   LaserEnd_Ext()
   LIN {X 9.720, Y 7.023, Z 94.350}
   LaserStart_Ext()
   LIN {X 9.720, Y -22.180, Z 94.350}
   LaserEnd_Ext()
   LIN {X 10.720, Y -19.592, Z 94.350}
   LaserStart_Ext()
   LIN {X 10.720, Y 0.002, Z 94.350}
   LaserEnd_Ext()
   LIN {X 5.886, Y -14.219, Z 95.200}
   LaserStart_Ext()
   LIN {X 6.069, Y -14.305, Z 95.200} C_DIS
   LIN {X 6.222, Y -14.503, Z 95.200} C_DIS
   LIN {X 7.618, Y -16.321, Z 95.200} C_DIS
   LIN {X 7.985, Y -18.449, Z 95.200} C_DIS
   LIN {X 7.977, Y -18.559, Z 95.200} C_DIS
   LIN {X 7.385, Y -20.644, Z 95.200} C_DIS
   LIN {X 5.903, Y -22.320, Z 95.200} C_DIS
   LIN {X 5.822, Y -22.379, Z 95.200} C_DIS
   LIN {X 3.889, Y -23.196, Z 95.200} C_DIS
   LIN {X 2.561, Y -23.174, Z 95.200} C_DIS
   LIN {X 1.827, Y -23.160, Z 95.200} C_DIS
   LIN {X 0.884, Y -22.715, Z 95.200} C_DIS
   LIN {X -0.043, Y -22.280, Z 95.200} C_DIS
   LIN {X -0.599, Y -21.642, Z 95.200} C_DIS
   LIN {X -1.407, Y -20.706, Z 95.200} C_DIS
   LIN {X -1.753, Y -19.527, Z 95.200} C_DIS
   LIN {X -1.997, Y -18.705, Z 95.200} C_DIS
   LIN {X -1.693, Y -17.374, Z 95.200} C_DIS
   LIN {X -1.338, Y -15.799, Z 95.200} C_DIS
   LIN {X -0.761, Y -15.153, Z 95.200} C_DIS
   LIN {X 0.076, Y -14.226, Z 95.200} C_DIS
   LIN {X 1.728, Y -13.494, Z 95.200} C_DIS
   LIN {X 1.983, Y -13.382, Z 95.200} C_DIS
   LIN {X 2.192, Y -13.383, Z 95.200} C_DIS
   LIN {X 4.149, Y -13.393, Z 95.200} C_DIS
   LIN {X 5.886, Y -14.219, Z 95.200}
   LaserEnd_Ext()
   LIN {X -5.498, Y -20.746, Z 95.200}
   LaserStart_Ext()
   LIN {X -6.019, Y -18.561, Z 95.200} C_DIS
   LIN {X -5.683, Y -16.347, Z 95.200} C_DIS
   LIN {X -5.539, Y -15.427, Z 95.200} C_DIS
   LIN {X -5.305, Y -14.701, Z 95.200} C_DIS
   LIN {X -4.631, Y -12.568, Z 95.200} C_DIS
   LIN {X -3.664, Y -8.937, Z 95.200} C_DIS
   LIN {X -3.638, Y -8.835, Z 95.200} C_DIS
   LIN {X -2.885, Y -5.203, Z 95.200} C_DIS
   LIN {X -2.566, Y -3.350, Z 95.200} C_DIS
   LIN {X -2.304, Y -1.628, Z 95.200} C_DIS
   LIN {X -2.221, Y -0.926, Z 95.200} C_DIS
   LIN {X -2.134, Y -0.229, Z 95.200} C_DIS
   LIN {X -1.879, Y 2.505, Z 95.200} C_DIS
   LIN {X -1.732, Y 6.473, Z 95.200} C_DIS
   LIN {X -1.751, Y 11.457, Z 95.200} C_DIS
   LIN {X -2.156, Y 15.764, Z 95.200} C_DIS
   LIN {X -3.665, Y 24.816, Z 95.200} C_DIS
   LIN {X -3.882, Y 25.807, Z 95.200} C_DIS
   LIN {X -4.262, Y 27.109, Z 95.200} C_DIS
   LIN {X -5.179, Y 30.344, Z 95.200} C_DIS
   LIN {X -6.003, Y 32.721, Z 95.200} C_DIS
   LIN {X -6.559, Y 34.208, Z 95.200} C_DIS
   LIN {X -7.213, Y 35.871, Z 95.200} C_DIS
   LIN {X -7.302, Y 36.098, Z 95.200} C_DIS
   LIN {X -7.368, Y 36.249, Z 95.200} C_DIS
   LIN {X -8.249, Y 38.271, Z 95.200} C_DIS
   LIN {X -8.844, Y 39.539, Z 95.200} C_DIS
   LIN {X -8.928, Y 39.719, Z 95.200} C_DIS
   LIN {X -9.034, Y 39.937, Z 95.200} C_DIS
   LIN {X -9.471, Y 40.846, Z 95.200} C_DIS
   LIN {X -9.752, Y 41.728, Z 95.200} C_DIS
   LIN {X -9.875, Y 42.116, Z 95.200} C_DIS
   LIN {X -9.856, Y 42.526, Z 95.200} C_DIS
   LIN {X -9.820, Y 43.494, Z 95.200} C_DIS
   LIN {X -9.382, Y 44.438, Z 95.200} C_DIS
   LIN {X -9.073, Y 45.084, Z 95.200} C_DIS
   LIN {X -8.537, Y 45.414, Z 95.200} C_DIS
   LIN {X -6.714, Y 46.543, Z 95.200} C_DIS
   LIN {X -6.039, Y 46.527, Z 95.200} C_DIS
   LIN {X -4.970, Y 46.499, Z 95.200} C_DIS
   LIN {X -3.550, Y 45.789, Z 95.200} C_DIS
   LIN {X -3.415, Y 45.721, Z 95.200} C_DIS
   LIN {X -2.455, Y 44.605, Z 95.200} C_DIS
   LIN {X -1.797, Y 43.427, Z 95.200} C_DIS
   LIN {X -1.731, Y 43.308, Z 95.200} C_DIS
   LIN {X -1.605, Y 43.078, Z 95.200} C_DIS
   LIN {X -0.809, Y 41.619, Z 95.200} C_DIS
   LIN {X -0.065, Y 40.182, Z 95.200} C_DIS
   LIN {X 0.629, Y 38.834, Z 95.200} C_DIS
   LIN {X 0.808, Y 38.450, Z 95.200} C_DIS
   LIN {X 3.585, Y 32.416, Z 95.200} C_DIS
   LIN {X 4.111, Y 31.131, Z 95.200} C_DIS
   LIN {X 5.388, Y 27.470, Z 95.200} C_DIS
   LIN {X 6.945, Y 23.293, Z 95.200} C_DIS
   LIN {X 7.649, Y 21.147, Z 95.200} C_DIS
   LIN {X 9.644, Y 13.265, Z 95.200} C_DIS
   LIN {X 9.975, Y 11.963, Z 95.200} C_DIS
   LIN {X 10.184, Y 10.632, Z 95.200} C_DIS
   LIN {X 11.571, Y 2.143, Z 95.200} C_DIS
   LIN {X 11.760, Y 0.223, Z 95.200} C_DIS
   LIN {X 12.012, Y -2.890, Z 95.200} C_DIS
   LIN {X 12.109, Y -4.088, Z 95.200} C_DIS
   LIN {X 12.241, Y -7.692, Z 95.200} C_DIS
   LIN {X 12.287, Y -8.871, Z 95.200} C_DIS
   LIN {X 12.289, Y -9.206, Z 95.200} C_DIS
   LIN {X 12.281, Y -12.675, Z 95.200} C_DIS
   LIN {X 12.228, Y -14.437, Z 95.200} C_DIS
   LIN {X 12.185, Y -15.633, Z 95.200} C_DIS
   LIN {X 12.037, Y -18.085, Z 95.200} C_DIS
   LIN {X 11.990, Y -18.889, Z 95.200} C_DIS
   LIN {X 11.897, Y -19.276, Z 95.200} C_DIS
   LIN {X 11.284, Y -21.766, Z 95.200} C_DIS
   LIN {X 9.658, Y -24.025, Z 95.200} C_DIS
   LIN {X 8.896, Y -25.053, Z 95.200} C_DIS
   LIN {X 5.588, Y -26.867, Z 95.200} C_DIS
   LIN {X 5.471, Y -26.932, Z 95.200} C_DIS
   LIN {X 5.278, Y -26.929, Z 95.200} C_DIS
   LIN {X -0.325, Y -26.687, Z 95.200} C_DIS
   LIN {X -1.234, Y -26.081, Z 95.200} C_DIS
   LIN {X -3.494, Y -24.588, Z 95.200} C_DIS
   LIN {X -4.454, Y -23.208, Z 95.200} C_DIS
   LIN {X -5.166, Y -22.172, Z 95.200} C_DIS
   LIN {X -5.498, Y -20.746, Z 95.200}
   LaserEnd_Ext()
   LIN {X -0.513, Y -25.360, Z 95.200}
   LaserStart_Ext()
   LIN {X 6.256, Y -25.360, Z 95.200}
   LaserEnd_Ext()
   LIN {X 8.080, Y -24.360, Z 95.200}
   LaserStart_Ext()
   LIN {X -2.025, Y -24.360, Z 95.200}
   LaserEnd_Ext()
   LIN {X -3.130, Y -23.360, Z 95.200}
   LaserStart_Ext()
   LIN {X -0.096, Y -23.360, Z 95.200}
   LaserEnd_Ext()
   LIN {X 6.069, Y -23.360, Z 95.200}
   LaserStart_Ext()
   LIN {X 8.904, Y -23.360, Z 95.200}
   LaserEnd_Ext()
   LIN {X 9.624, Y -22.360, Z 95.200}
   LaserStart_Ext()
   LIN {X 7.202, Y -22.360, Z 95.200}
   LaserEnd_Ext()
   LIN {X -1.299, Y -22.360, Z 95.200}
   LaserStart_Ext()
   LIN {X -3.823, Y -22.360, Z 95.200}
   LaserEnd_Ext()
   LIN {X -4.328, Y -21.360, Z 95.200}
   LaserStart_Ext()
   LIN {X -2.164, Y -21.360, Z 95.200}
   LaserEnd_Ext()
   LIN {X 8.087, Y -21.360, Z 95.200}
   LaserStart_Ext()
   LIN {X 10.344, Y -21.360, Z 95.200}
   LaserEnd_Ext()
   LIN {X 10.600, Y -20.360, Z 95.200}
   LaserStart_Ext()
   LIN {X 8.505, Y -20.360, Z 95.200}
   LaserEnd_Ext()
   LIN {X -2.551, Y -20.360, Z 95.200}
   LaserStart_Ext()
   LIN {X -4.562, Y -20.360, Z 95.200}
   LaserEnd_Ext()
   LIN {X -4.800, Y -19.360, Z 95.200}
   LaserStart_Ext()
   LIN {X -2.846, Y -19.360, Z 95.200}
   LaserEnd_Ext()
   LIN {X 8.789, Y -19.360, Z 95.200}
   LaserStart_Ext()
   LIN {X 10.847, Y -19.360, Z 95.200}
   LaserEnd_Ext()
   LIN {X 11.019, Y -18.360, Z 95.200}
   LaserStart_Ext()
   LIN {X 8.983, Y -18.360, Z 95.200}
   LaserEnd_Ext()
   LIN {X -2.944, Y -18.360, Z 95.200}
   LaserStart_Ext()
   LIN {X -4.977, Y -18.360, Z 95.200}
   LaserEnd_Ext()
   LIN {X -4.825, Y -17.360, Z 95.200}
   LaserStart_Ext()
   LIN {X -2.716, Y -17.360, Z 95.200}
   LaserEnd_Ext()
   LIN {X 8.812, Y -17.360, Z 95.200}
   LaserStart_Ext()
   LIN {X 11.079, Y -17.360, Z 95.200}
   LaserEnd_Ext()
   LIN {X 11.139, Y -16.360, Z 95.200}
   LaserStart_Ext()
   LIN {X 8.639, Y -16.360, Z 95.200}
   LaserEnd_Ext()
   LIN {X -2.489, Y -16.360, Z 95.200}
   LaserStart_Ext()
   LIN {X -4.673, Y -16.360, Z 95.200}
   LaserEnd_Ext()
   LIN {X -4.467, Y -15.360, Z 95.200}
   LaserStart_Ext()
   LIN {X -2.235, Y -15.360, Z 95.200}
   LaserEnd_Ext()
   LIN {X 8.140, Y -15.360, Z 95.200}
   LaserStart_Ext()
   LIN {X 11.194, Y -15.360, Z 95.200}
   LaserEnd_Ext()
   LIN {X 11.230, Y -14.360, Z 95.200}
   LaserStart_Ext()
   LIN {X 7.373, Y -14.360, Z 95.200}
   LaserEnd_Ext()
   LIN {X -1.392, Y -14.360, Z 95.200}
   LaserStart_Ext()
   LIN {X -4.149, Y -14.360, Z 95.200}
   LaserEnd_Ext()
   LIN {X -3.833, Y -13.360, Z 95.200}
   LaserStart_Ext()
   LIN {X -0.425, Y -13.360, Z 95.200}
   LaserEnd_Ext()
   LIN {X 6.409, Y -13.360, Z 95.200}
   LaserStart_Ext()
   LIN {X 11.260, Y -13.360, Z 95.200}
   LaserEnd_Ext()
   LIN {X 11.282, Y -12.360, Z 95.200}
   LaserStart_Ext()
   LIN {X -3.541, Y -12.360, Z 95.200}
   LaserEnd_Ext()
   LIN {X -3.274, Y -11.360, Z 95.200}
   LaserStart_Ext()
   LIN {X 11.284, Y -11.360, Z 95.200}
   LaserEnd_Ext()
   LIN {X 11.286, Y -10.360, Z 95.200}
   LaserStart_Ext()
   LIN {X -3.008, Y -10.360, Z 95.200}
   LaserEnd_Ext()
   LIN {X -2.742, Y -9.360, Z 95.200}
   LaserStart_Ext()
   LIN {X 11.289, Y -9.360, Z 95.200}
   LaserEnd_Ext()
   LIN {X 11.267, Y -8.360, Z 95.200}
   LaserStart_Ext()
   LIN {X -2.518, Y -8.360, Z 95.200}
   LaserEnd_Ext()
   LIN {X -2.311, Y -7.360, Z 95.200}
   LaserStart_Ext()
   LIN {X 11.228, Y -7.360, Z 95.200}
   LaserEnd_Ext()
   LIN {X 11.192, Y -6.360, Z 95.200}
   LaserStart_Ext()
   LIN {X -2.104, Y -6.360, Z 95.200}
   LaserEnd_Ext()
   LIN {X -1.897, Y -5.360, Z 95.200}
   LaserStart_Ext()
   LIN {X 11.155, Y -5.360, Z 95.200}
   LaserEnd_Ext()
   LIN {X 11.118, Y -4.360, Z 95.200}
   LaserStart_Ext()
   LIN {X -1.725, Y -4.360, Z 95.200}
   LaserEnd_Ext()
   LIN {X -1.556, Y -3.360, Z 95.200}
   LaserStart_Ext()
   LIN {X 11.047, Y -3.360, Z 95.200}
   LaserEnd_Ext()
   LIN {X 10.966, Y -2.360, Z 95.200}
   LaserStart_Ext()
   LIN {X -1.404, Y -2.360, Z 95.200}
   LaserEnd_Ext()
   LIN {X -1.265, Y -1.360, Z 95.200}
   LaserStart_Ext()
   LIN {X 10.885, Y -1.360, Z 95.200}
   LaserEnd_Ext()
   LIN {X 10.804, Y -0.360, Z 95.200}
   LaserStart_Ext()
   LIN {X -1.142, Y -0.360, Z 95.200}
   LaserEnd_Ext()
   LIN {X -1.048, Y 0.640, Z 95.200}
   LaserStart_Ext()
   LIN {X 10.714, Y 0.640, Z 95.200}
   LaserEnd_Ext()
   LIN {X 10.615, Y 1.640, Z 95.200}
   LaserStart_Ext()
   LIN {X -0.955, Y 1.640, Z 95.200}
   LaserEnd_Ext()
   LIN {X -0.873, Y 2.640, Z 95.200}
   LaserStart_Ext()
   LIN {X 10.476, Y 2.640, Z 95.200}
   LaserEnd_Ext()
   LIN {X 10.313, Y 3.640, Z 95.200}
   LaserStart_Ext()
   LIN {X -0.836, Y 3.640, Z 95.200}
   LaserEnd_Ext()
   LIN {X -0.799, Y 4.640, Z 95.200}
   LaserStart_Ext()
   LIN {X 10.150, Y 4.640, Z 95.200}
   LaserEnd_Ext()
   LIN {X 9.986, Y 5.640, Z 95.200}
   LaserStart_Ext()
   LIN {X -0.762, Y 5.640, Z 95.200}
   LaserEnd_Ext()
   LIN {X -0.733, Y 6.640, Z 95.200}
   LaserStart_Ext()
   LIN {X 9.823, Y 6.640, Z 95.200}
   LaserEnd_Ext()
   LIN {X 9.660, Y 7.640, Z 95.200}
   LaserStart_Ext()
   LIN {X -0.736, Y 7.640, Z 95.200}
   LaserEnd_Ext()
   LIN {X -0.740, Y 8.640, Z 95.200}
   LaserStart_Ext()
   LIN {X 9.496, Y 8.640, Z 95.200}
   LaserEnd_Ext()
   LIN {X 9.333, Y 9.640, Z 95.200}
   LaserStart_Ext()
   LIN {X -0.744, Y 9.640, Z 95.200}
   LaserEnd_Ext()
   LIN {X -0.748, Y 10.640, Z 95.200}
   LaserStart_Ext()
   LIN {X 9.171, Y 10.640, Z 95.200}
   LaserEnd_Ext()
   LIN {X 9.014, Y 11.640, Z 95.200}
   LaserStart_Ext()
   LIN {X -0.764, Y 11.640, Z 95.200}
   LaserEnd_Ext()
   LIN {X -0.858, Y 12.640, Z 95.200}
   LaserStart_Ext()
   LIN {X 8.771, Y 12.640, Z 95.200}
   LaserEnd_Ext()
   LIN {X 8.517, Y 13.640, Z 95.200}
   LaserStart_Ext()
   LIN {X -0.952, Y 13.640, Z 95.200}
   LaserEnd_Ext()
   LIN {X -1.046, Y 14.640, Z 95.200}
   LaserStart_Ext()
   LIN {X 8.264, Y 14.640, Z 95.200}
   LaserEnd_Ext()
   LIN {X 8.011, Y 15.640, Z 95.200}
   LaserStart_Ext()
   LIN {X -1.140, Y 15.640, Z 95.200}
   LaserEnd_Ext()
   LIN {X -1.288, Y 16.640, Z 95.200}
   LaserStart_Ext()
   LIN {X 7.758, Y 16.640, Z 95.200}
   LaserEnd_Ext()
   LIN {X 7.505, Y 17.640, Z 95.200}
   LaserStart_Ext()
   LIN {X -1.455, Y 17.640, Z 95.200}
   LaserEnd_Ext()
   LIN {X -1.622, Y 18.640, Z 95.200}
   LaserStart_Ext()
   LIN {X 7.252, Y 18.640, Z 95.200}
   LaserEnd_Ext()
   LIN {X 6.999, Y 19.640, Z 95.200}
   LaserStart_Ext()
   LIN {X -1.789, Y 19.640, Z 95.200}
   LaserEnd_Ext()
   LIN {X -1.955, Y 20.640, Z 95.200}
   LaserStart_Ext()
   LIN {X 6.746, Y 20.640, Z 95.200}
   LaserEnd_Ext()
   LIN {X 6.435, Y 21.640, Z 95.200}
   LaserStart_Ext()
   LIN {X -2.122, Y 21.640, Z 95.200}
   LaserEnd_Ext()
   LIN {X -2.289, Y 22.640, Z 95.200}
   LaserStart_Ext()
   LIN {X 6.106, Y 22.640, Z 95.200}
   LaserEnd_Ext()
   LIN {X 5.748, Y 23.640, Z 95.200}
   LaserStart_Ext()
   LIN {X -2.455, Y 23.640, Z 95.200}
   LaserEnd_Ext()
   LIN {X -2.622, Y 24.640, Z 95.200}
   LaserStart_Ext()
   LIN {X 5.375, Y 24.640, Z 95.200}
   LaserEnd_Ext()
   LIN {X 5.003, Y 25.640, Z 95.200}
   LaserStart_Ext()
   LIN {X -2.822, Y 25.640, Z 95.200}
   LaserEnd_Ext()
   LIN {X -3.083, Y 26.640, Z 95.200}
   LaserStart_Ext()
   LIN {X 4.630, Y 26.640, Z 95.200}
   LaserEnd_Ext()
   LIN {X 4.270, Y 27.640, Z 95.200}
   LaserStart_Ext()
   LIN {X -3.373, Y 27.640, Z 95.200}
   LaserEnd_Ext()
   LIN {X -3.657, Y 28.640, Z 95.200}
   LaserStart_Ext()
   LIN {X 3.921, Y 28.640, Z 95.200}
   LaserEnd_Ext()
   LIN {X 3.572, Y 29.640, Z 95.200}
   LaserStart_Ext()
   LIN {X -3.940, Y 29.640, Z 95.200}
   LaserEnd_Ext()
   LIN {X -4.225, Y 30.640, Z 95.200}
   LaserStart_Ext()
   LIN {X 3.224, Y 30.640, Z 95.200}
   LaserEnd_Ext()
   LIN {X 2.822, Y 31.640, Z 95.200}
   LaserStart_Ext()
   LIN {X -4.570, Y 31.640, Z 95.200}
   LaserEnd_Ext()
   LIN {X -4.917, Y 32.640, Z 95.200}
   LaserStart_Ext()
   LIN {X 2.381, Y 32.640, Z 95.200}
   LaserEnd_Ext()
   LIN {X 1.921, Y 33.640, Z 95.200}
   LaserStart_Ext()
   LIN {X -5.279, Y 33.640, Z 95.200}
   LaserEnd_Ext()
   LIN {X -5.654, Y 34.640, Z 95.200}
   LaserStart_Ext()
   LIN {X 1.461, Y 34.640, Z 95.200}
   LaserEnd_Ext()
   LIN {X 1.000, Y 35.640, Z 95.200}
   LaserStart_Ext()
   LIN {X -6.048, Y 35.640, Z 95.200}
   LaserEnd_Ext()
   LIN {X -6.447, Y 36.640, Z 95.200}
   LaserStart_Ext()
   LIN {X 0.540, Y 36.640, Z 95.200}
   LaserEnd_Ext()
   LIN {X 0.080, Y 37.640, Z 95.200}
   LaserStart_Ext()
   LIN {X -6.883, Y 37.640, Z 95.200}
   LaserEnd_Ext()
   LIN {X -7.319, Y 38.640, Z 95.200}
   LaserStart_Ext()
   LIN {X -0.396, Y 38.640, Z 95.200}
   LaserEnd_Ext()
   LIN {X -0.911, Y 39.640, Z 95.200}
   LaserStart_Ext()
   LIN {X -7.787, Y 39.640, Z 95.200}
   LaserEnd_Ext()
   LIN {X -8.262, Y 40.640, Z 95.200}
   LaserStart_Ext()
   LIN {X -1.428, Y 40.640, Z 95.200}
   LaserEnd_Ext()
   LIN {X -1.960, Y 41.640, Z 95.200}
   LaserStart_Ext()
   LIN {X -8.674, Y 41.640, Z 95.200}
   LaserEnd_Ext()
   LIN {X -8.851, Y 42.640, Z 95.200}
   LaserStart_Ext()
   LIN {X -2.506, Y 42.640, Z 95.200}
   LaserEnd_Ext()
   LIN {X -3.061, Y 43.640, Z 95.200}
   LaserStart_Ext()
   LIN {X -8.650, Y 43.640, Z 95.200}
   LaserEnd_Ext()
   LIN {X -7.888, Y 44.640, Z 95.200}
   LaserStart_Ext()
   LIN {X -3.803, Y 44.640, Z 95.200}
   LaserEnd_Ext()
   LIN {X 7.418, Y -20.676, Z 96.050}
   LaserStart_Ext()
   LIN {X 7.313, Y -20.795, Z 96.050} C_DIS
   LIN {X 5.955, Y -22.298, Z 96.050} C_DIS
   LIN {X 4.796, Y -22.790, Z 96.050} C_DIS
   LIN {X 3.975, Y -23.138, Z 96.050} C_DIS
   LIN {X 2.680, Y -23.116, Z 96.050} C_DIS
   LIN {X 1.920, Y -23.105, Z 96.050} C_DIS
   LIN {X 1.422, Y -22.874, Z 96.050} C_DIS
   LIN {X 0.048, Y -22.229, Z 96.050} C_DIS
   LIN {X -1.160, Y -20.841, Z 96.050} C_DIS
   LIN {X -1.320, Y -20.658, Z 96.050} C_DIS
   LIN {X -1.384, Y -20.446, Z 96.050} C_DIS
   LIN {X -1.914, Y -18.659, Z 96.050} C_DIS
   LIN {X -1.369, Y -16.270, Z 96.050} C_DIS
   LIN {X -1.243, Y -15.719, Z 96.050} C_DIS
   LIN {X -0.908, Y -15.348, Z 96.050} C_DIS
   LIN {X 0.156, Y -14.168, Z 96.050} C_DIS
   LIN {X 1.141, Y -13.732, Z 96.050} C_DIS
   LIN {X 2.053, Y -13.326, Z 96.050} C_DIS
   LIN {X 3.470, Y -13.328, Z 96.050} C_DIS
   LIN {X 4.219, Y -13.332, Z 96.050} C_DIS
   LIN {X 4.753, Y -13.586, Z 96.050} C_DIS
   LIN {X 6.141, Y -14.240, Z 96.050} C_DIS
   LIN {X 7.304, Y -15.743, Z 96.050} C_DIS
   LIN {X 7.695, Y -16.252, Z 96.050} C_DIS
   LIN {X 7.803, Y -16.879, Z 96.050} C_DIS
   LIN {X 8.076, Y -18.429, Z 96.050} C_DIS
   LIN {X 7.460, Y -20.527, Z 96.050} C_DIS
   LIN {X 7.418, Y -20.676, Z 96.050}
   LaserEnd_Ext()
   LIN {X -8.287, Y 38.272, Z 96.050}
   LaserStart_Ext()
   LIN {X -7.348, Y 36.132, Z 96.050} C_DIS
   LIN {X -6.974, Y 35.180, Z 96.050} C_DIS
   LIN {X -5.639, Y 31.611, Z 96.050} C_DIS
   LIN {X -5.201, Y 30.347, Z 96.050} C_DIS
   LIN {X -4.714, Y 28.628, Z 96.050} C_DIS
   LIN {X -3.924, Y 25.925, Z 96.050} C_DIS
   LIN {X -3.475, Y 23.867, Z 96.050} C_DIS
   LIN {X -2.206, Y 16.260, Z 96.050} C_DIS
   LIN {X -1.721, Y 11.097, Z 96.050} C_DIS
   LIN {X -1.704, Y 6.823, Z 96.050} C_DIS
   LIN {X -1.878, Y 2.146, Z 96.050} C_DIS
   LIN {X -2.093, Y -0.165, Z 96.050} C_DIS
   LIN {X -2.167, Y -0.755, Z 96.050} C_DIS
   LIN {X -2.285, Y -1.759, Z 96.050} C_DIS
   LIN {X -2.445, Y -2.806, Z 96.050} C_DIS
   LIN {X -2.997, Y -6.017, Z 96.050} C_DIS
   LIN {X -3.487, Y -8.375, Z 96.050} C_DIS
   LIN {X -3.992, Y -10.385, Z 96.050} C_DIS
   LIN {X -4.557, Y -12.506, Z 96.050} C_DIS
   LIN {X -5.255, Y -14.716, Z 96.050} C_DIS
   LIN {X -5.465, Y -15.389, Z 96.050} C_DIS
   LIN {X -5.553, Y -15.995, Z 96.050} C_DIS
   LIN {X -5.937, Y -18.524, Z 96.050} C_DIS
   LIN {X -5.120, Y -21.953, Z 96.050} C_DIS
   LIN {X -5.076, Y -22.134, Z 96.050} C_DIS
   LIN {X -4.986, Y -22.262, Z 96.050} C_DIS
   LIN {X -3.398, Y -24.545, Z 96.050} C_DIS
   LIN {X -0.974, Y -26.147, Z 96.050} C_DIS
   LIN {X -0.221, Y -26.638, Z 96.050} C_DIS
   LIN {X 0.213, Y -26.717, Z 96.050} C_DIS
   LIN {X 4.984, Y -26.957, Z 96.050} C_DIS
   LIN {X 5.688, Y -26.829, Z 96.050} C_DIS
   LIN {X 8.909, Y -25.025, Z 96.050} C_DIS
   LIN {X 9.026, Y -24.954, Z 96.050} C_DIS
   LIN {X 9.240, Y -24.652, Z 96.050} C_DIS
   LIN {X 11.374, Y -21.688, Z 96.050} C_DIS
   LIN {X 11.683, Y -20.434, Z 96.050} C_DIS
   LIN {X 12.072, Y -18.810, Z 96.050} C_DIS
   LIN {X 12.258, Y -15.609, Z 96.050} C_DIS
   LIN {X 12.263, Y -15.475, Z 96.050} C_DIS
   LIN {X 12.349, Y -12.595, Z 96.050} C_DIS
   LIN {X 12.354, Y -10.415, Z 96.050} C_DIS
   LIN {X 12.346, Y -8.791, Z 96.050} C_DIS
   LIN {X 12.172, Y -4.347, Z 96.050} C_DIS
   LIN {X 12.155, Y -3.988, Z 96.050} C_DIS
   LIN {X 11.862, Y -0.359, Z 96.050} C_DIS
   LIN {X 11.621, Y 2.083, Z 96.050} C_DIS
   LIN {X 10.107, Y 11.350, Z 96.050} C_DIS
   LIN {X 10.032, Y 11.811, Z 96.050} C_DIS
   LIN {X 9.888, Y 12.387, Z 96.050} C_DIS
   LIN {X 7.731, Y 20.909, Z 96.050} C_DIS
   LIN {X 6.836, Y 23.635, Z 96.050} C_DIS
   LIN {X 4.858, Y 28.942, Z 96.050} C_DIS
   LIN {X 4.054, Y 31.249, Z 96.050} C_DIS
   LIN {X 3.722, Y 32.059, Z 96.050} C_DIS
   LIN {X 1.159, Y 37.626, Z 96.050} C_DIS
   LIN {X 0.617, Y 38.806, Z 96.050} C_DIS
   LIN {X -0.122, Y 40.227, Z 96.050} C_DIS
   LIN {X -0.872, Y 41.675, Z 96.050} C_DIS
   LIN {X -1.122, Y 42.135, Z 96.050} C_DIS
   LIN {X -1.794, Y 43.357, Z 96.050} C_DIS
   LIN {X -2.507, Y 44.626, Z 96.050} C_DIS
   LIN {X -3.482, Y 45.765, Z 96.050} C_DIS
   LIN {X -4.742, Y 46.391, Z 96.050} C_DIS
   LIN {X -5.040, Y 46.539, Z 96.050} C_DIS
   LIN {X -5.608, Y 46.551, Z 96.050} C_DIS
   LIN {X -6.785, Y 46.578, Z 96.050} C_DIS
   LIN {X -7.367, Y 46.217, Z 96.050} C_DIS
   LIN {X -9.123, Y 45.135, Z 96.050} C_DIS
   LIN {X -9.539, Y 44.263, Z 96.050} C_DIS
   LIN {X -9.867, Y 43.593, Z 96.050} C_DIS
   LIN {X -9.904, Y 42.944, Z 96.050} C_DIS
   LIN {X -9.940, Y 42.181, Z 96.050} C_DIS
   LIN {X -9.722, Y 41.496, Z 96.050} C_DIS
   LIN {X -9.527, Y 40.875, Z 96.050} C_DIS
   LIN {X -9.344, Y 40.499, Z 96.050} C_DIS
   LIN {X -8.982, Y 39.749, Z 96.050} C_DIS
   LIN {X -8.308, Y 38.319, Z 96.050}
   LaserEnd_Ext()
   LIN {X 10.602, Y 2.117, Z 96.050}
   LaserStart_Ext()
   LIN {X 10.602, Y -20.641, Z 96.050}
   LaserEnd_Ext()
   LIN {X 9.602, Y -22.438, Z 96.050}
   LaserStart_Ext()
   LIN {X 9.602, Y 8.241, Z 96.050}
   LaserEnd_Ext()
   LIN {X 8.602, Y 13.391, Z 96.050}
   LaserStart_Ext()
   LIN {X 8.602, Y -15.834, Z 96.050}
   LaserEnd_Ext()
   LIN {X 8.602, Y -20.187, Z 96.050}
   LaserStart_Ext()
   LIN {X 8.602, Y -23.827, Z 96.050}
   LaserEnd_Ext()
   LIN {X 7.602, Y -24.611, Z 96.050}
   LaserStart_Ext()
   LIN {X 7.602, Y -21.966, Z 96.050}
   LaserEnd_Ext()
   LIN {X 7.602, Y -14.494, Z 96.050}
   LaserStart_Ext()
   LIN {X 7.602, Y 17.343, Z 96.050}
   LaserEnd_Ext()
   LIN {X 6.602, Y 21.142, Z 96.050}
   LaserStart_Ext()
   LIN {X 6.602, Y -13.353, Z 96.050}
   LaserEnd_Ext()
   LIN {X 6.602, Y -23.059, Z 96.050}
   LaserStart_Ext()
   LIN {X 6.602, Y -25.171, Z 96.050}
   LaserEnd_Ext()
   LIN {X 5.602, Y -25.732, Z 96.050}
   LaserStart_Ext()
   LIN {X 5.602, Y -23.534, Z 96.050}
   LaserEnd_Ext()
   LIN {X 5.602, Y -12.880, Z 96.050}
   LaserStart_Ext()
   LIN {X 5.602, Y 24.083, Z 96.050}
   LaserEnd_Ext()
   LIN {X 4.602, Y 26.766, Z 96.050}
   LaserStart_Ext()
   LIN {X 4.602, Y -12.410, Z 96.050}
   LaserEnd_Ext()
   LIN {X 4.602, Y -23.958, Z 96.050}
   LaserStart_Ext()
   LIN {X 4.602, Y -25.937, Z 96.050}
   LaserEnd_Ext()
   LIN {X 3.602, Y -25.887, Z 96.050}
   LaserStart_Ext()
   LIN {X 3.602, Y -24.132, Z 96.050}
   LaserEnd_Ext()
   LIN {X 3.602, Y -12.329, Z 96.050}
   LaserStart_Ext()
   LIN {X 3.602, Y 29.508, Z 96.050}
   LaserEnd_Ext()
   LIN {X 2.602, Y 32.101, Z 96.050}
   LaserStart_Ext()
   LIN {X 2.602, Y -12.327, Z 96.050}
   LaserEnd_Ext()
   LIN {X 2.602, Y -24.115, Z 96.050}
   LaserStart_Ext()
   LIN {X 2.602, Y -25.836, Z 96.050}
   LaserEnd_Ext()
   LIN {X 1.602, Y -25.786, Z 96.050}
   LaserStart_Ext()
   LIN {X 1.602, Y -24.053, Z 96.050}
   LaserEnd_Ext()
   LIN {X 1.602, Y -12.432, Z 96.050}
   LaserStart_Ext()
   LIN {X 1.602, Y 34.274, Z 96.050}
   LaserEnd_Ext()
   LIN {X 0.602, Y 36.446, Z 96.050}
   LaserStart_Ext()
   LIN {X 0.602, Y -12.877, Z 96.050}
   LaserEnd_Ext()
   LIN {X 0.602, Y -23.594, Z 96.050}
   LaserStart_Ext()
   LIN {X 0.602, Y -25.736, Z 96.050}
   LaserEnd_Ext()
   LIN {X -0.398, Y -25.329, Z 96.050}
   LaserStart_Ext()
   LIN {X -0.398, Y -23.123, Z 96.050}
   LaserEnd_Ext()
   LIN {X -0.398, Y -13.338, Z 96.050}
   LaserStart_Ext()
   LIN {X -0.398, Y 38.591, Z 96.050}
   LaserEnd_Ext()
   LIN {X -1.398, Y 40.517, Z 96.050}
   LaserStart_Ext()
   LIN {X -1.398, Y 17.492, Z 96.050}
   LaserEnd_Ext()
   LIN {X -1.398, Y -2.576, Z 96.050}
   LaserStart_Ext()
   LIN {X -1.398, Y -14.398, Z 96.050}
   LaserEnd_Ext()
   LIN {X -1.398, Y -22.091, Z 96.050}
   LaserStart_Ext()
   LIN {X -1.398, Y -24.668, Z 96.050}
   LaserEnd_Ext()
   LIN {X -2.398, Y -24.007, Z 96.050}
   LaserStart_Ext()
   LIN {X -2.398, Y -20.543, Z 96.050}
   LaserEnd_Ext()
   LIN {X -2.398, Y -16.286, Z 96.050}
   LaserStart_Ext()
   LIN {X -2.398, Y -8.051, Z 96.050}
   LaserEnd_Ext()
   LIN {X -2.398, Y 23.490, Z 96.050}
   LaserStart_Ext()
   LIN {X -2.398, Y 42.380, Z 96.050}
   LaserEnd_Ext()
   LIN {X -3.398, Y 44.137, Z 96.050}
   LaserStart_Ext()
   LIN {X -3.398, Y 27.691, Z 96.050}
   LaserEnd_Ext()
   LIN {X -3.398, Y -12.041, Z 96.050}
   LaserStart_Ext()
   LIN {X -3.398, Y -22.793, Z 96.050}
   LaserEnd_Ext()
   LIN {X -4.398, Y -20.667, Z 96.050}
   LaserStart_Ext()
   LIN {X -4.398, Y -15.327, Z 96.050}
   LaserEnd_Ext()
   LIN {X -4.398, Y 31.084, Z 96.050}
   LaserStart_Ext()
   LIN {X -4.398, Y 45.103, Z 96.050}
   LaserEnd_Ext()
   LIN {X -5.398, Y 45.546, Z 96.050}
   LaserStart_Ext()
   LIN {X -5.398, Y 33.822, Z 96.050}
   LaserEnd_Ext()
   LIN {X -6.398, Y 36.449, Z 96.050}
   LaserStart_Ext()
   LIN {X -6.398, Y 45.569, Z 96.050}
   LaserEnd_Ext()
   LIN {X -7.398, Y 45.023, Z 96.050}
   LaserStart_Ext()
   LIN {X -7.398, Y 38.733, Z 96.050}
   LaserEnd_Ext()
   LIN {X -8.398, Y 40.839, Z 96.050}
   LaserStart_Ext()
   LIN {X -8.398, Y 44.332, Z 96.050}
   LaserEnd_Ext()
   LIN {X 3.573, Y -13.273, Z 96.900}
   LaserStart_Ext()
   LIN {X 4.290, Y -13.271, Z 96.900} C_DIS
   LIN {X 5.074, Y -13.637, Z 96.900} C_DIS
   LIN {X 6.213, Y -14.174, Z 96.900} C_DIS
   LIN {X 7.100, Y -15.321, Z 96.900} C_DIS
   LIN {X 7.772, Y -16.183, Z 96.900} C_DIS
   LIN {X 7.933, Y -17.082, Z 96.900} C_DIS
   LIN {X 8.158, Y -18.359, Z 96.900} C_DIS
   LIN {X 7.838, Y -19.449, Z 96.900} C_DIS
   LIN {X 7.497, Y -20.622, Z 96.900} C_DIS
   LIN {X 6.714, Y -21.492, Z 96.900} C_DIS
   LIN {X 6.039, Y -22.238, Z 96.900} C_DIS
   LIN {X 4.614, Y -22.843, Z 96.900} C_DIS
   LIN {X 4.072, Y -23.077, Z 96.900} C_DIS
   LIN {X 3.668, Y -23.074, Z 96.900} C_DIS
   LIN {X 2.014, Y -23.049, Z 96.900} C_DIS
   LIN {X 0.291, Y -22.250, Z 96.900} C_DIS
   LIN {X 0.139, Y -22.178, Z 96.900} C_DIS
   LIN {X 0.006, Y -22.025, Z 96.900} C_DIS
   LIN {X -1.232, Y -20.610, Z 96.900} C_DIS
   LIN {X -1.728, Y -18.962, Z 96.900} C_DIS
   LIN {X -1.832, Y -18.612, Z 96.900} C_DIS
   LIN {X -1.725, Y -18.145, Z 96.900} C_DIS
   LIN {X -1.158, Y -15.655, Z 96.900} C_DIS
   LIN {X 0.155, Y -14.202, Z 96.900} C_DIS
   LIN {X 0.237, Y -14.111, Z 96.900} C_DIS
   LIN {X 0.394, Y -14.041, Z 96.900} C_DIS
   LIN {X 2.123, Y -13.270, Z 96.900} C_DIS
   LIN {X 3.573, Y -13.273, Z 96.900}
   LaserEnd_Ext()
   LIN {X -1.691, Y 10.737, Z 96.900}
   LaserStart_Ext()
   LIN {X -1.677, Y 7.174, Z 96.900} C_DIS
   LIN {X -1.876, Y 1.787, Z 96.900} C_DIS
   LIN {X -2.052, Y -0.102, Z 96.900} C_DIS
   LIN {X -2.113, Y -0.583, Z 96.900} C_DIS
   LIN {X -2.267, Y -1.889, Z 96.900} C_DIS
   LIN {X -2.323, Y -2.262, Z 96.900} C_DIS
   LIN {X -3.110, Y -6.831, Z 96.900} C_DIS
   LIN {X -3.335, Y -7.915, Z 96.900} C_DIS
   LIN {X -4.320, Y -11.833, Z 96.900} C_DIS
   LIN {X -4.483, Y -12.444, Z 96.900} C_DIS
   LIN {X -4.684, Y -13.081, Z 96.900} C_DIS
   LIN {X -5.391, Y -15.351, Z 96.900} C_DIS
   LIN {X -5.689, Y -17.396, Z 96.900} C_DIS
   LIN {X -5.855, Y -18.488, Z 96.900} C_DIS
   LIN {X -5.502, Y -19.968, Z 96.900} C_DIS
   LIN {X -4.986, Y -22.094, Z 96.900} C_DIS
   LIN {X -3.926, Y -23.604, Z 96.900} C_DIS
   LIN {X -3.302, Y -24.503, Z 96.900} C_DIS
   LIN {X -2.348, Y -25.132, Z 96.900} C_DIS
   LIN {X -0.116, Y -26.589, Z 96.900} C_DIS
   LIN {X 1.167, Y -26.823, Z 96.900} C_DIS
   LIN {X 4.440, Y -26.988, Z 96.900} C_DIS
   LIN {X 5.941, Y -26.715, Z 96.900} C_DIS
   LIN {X 7.918, Y -25.607, Z 96.900} C_DIS
   LIN {X 9.153, Y -24.853, Z 96.900} C_DIS
   LIN {X 11.432, Y -21.654, Z 96.900} C_DIS
   LIN {X 12.154, Y -18.730, Z 96.900} C_DIS
   LIN {X 12.269, Y -16.742, Z 96.900} C_DIS
   LIN {X 12.335, Y -15.474, Z 96.900} C_DIS
   LIN {X 12.382, Y -13.693, Z 96.900} C_DIS
   LIN {X 12.417, Y -12.515, Z 96.900} C_DIS
   LIN {X 12.419, Y -11.624, Z 96.900} C_DIS
   LIN {X 12.405, Y -8.711, Z 96.900} C_DIS
   LIN {X 12.296, Y -5.915, Z 96.900} C_DIS
   LIN {X 12.195, Y -3.812, Z 96.900} C_DIS
   LIN {X 11.963, Y -0.941, Z 96.900} C_DIS
   LIN {X 11.671, Y 2.024, Z 96.900} C_DIS
   LIN {X 10.362, Y 10.038, Z 96.900} C_DIS
   LIN {X 10.111, Y 11.572, Z 96.900} C_DIS
   LIN {X 9.631, Y 13.485, Z 96.900} C_DIS
   LIN {X 7.813, Y 20.670, Z 96.900} C_DIS
   LIN {X 6.728, Y 23.977, Z 96.900} C_DIS
   LIN {X 4.329, Y 30.414, Z 96.900} C_DIS
   LIN {X 3.997, Y 31.367, Z 96.900} C_DIS
   LIN {X 3.860, Y 31.701, Z 96.900} C_DIS
   LIN {X 2.802, Y 33.999, Z 96.900} C_DIS
   LIN {X 0.585, Y 38.822, Z 96.900} C_DIS
   LIN {X -0.688, Y 41.270, Z 96.900} C_DIS
   LIN {X -0.931, Y 41.727, Z 96.900} C_DIS
   LIN {X -1.661, Y 43.049, Z 96.900} C_DIS
   LIN {X -1.856, Y 43.404, Z 96.900} C_DIS
   LIN {X -1.968, Y 43.603, Z 96.900} C_DIS
   LIN {X -2.585, Y 44.695, Z 96.900} C_DIS
   LIN {X -3.514, Y 45.766, Z 96.900} C_DIS
   LIN {X -3.633, Y 45.848, Z 96.900} C_DIS
   LIN {X -5.109, Y 46.578, Z 96.900} C_DIS
   LIN {X -6.120, Y 46.600, Z 96.900} C_DIS
   LIN {X -6.854, Y 46.613, Z 96.900} C_DIS
   LIN {X -8.585, Y 45.546, Z 96.900} C_DIS
   LIN {X -9.172, Y 45.185, Z 96.900} C_DIS
   LIN {X -9.532, Y 44.470, Z 96.900} C_DIS
   LIN {X -9.912, Y 43.691, Z 96.900} C_DIS
   LIN {X -9.953, Y 42.976, Z 96.900} C_DIS
   LIN {X -10.003, Y 42.249, Z 96.900} C_DIS
   LIN {X -9.790, Y 41.564, Z 96.900} C_DIS
   LIN {X -9.582, Y 40.904, Z 96.900} C_DIS
   LIN {X -9.183, Y 40.081, Z 96.900} C_DIS
   LIN {X -9.036, Y 39.779, Z 96.900} C_DIS
   LIN {X -8.917, Y 39.530, Z 96.900} C_DIS
   LIN {X -8.350, Y 38.334, Z 96.900} C_DIS
   LIN {X -7.406, Y 36.194, Z 96.900} C_DIS
   LIN {X -5.275, Y 30.501, Z 96.900} C_DIS
   LIN {X -5.223, Y 30.351, Z 96.900} C_DIS
   LIN {X -5.165, Y 30.146, Z 96.900} C_DIS
   LIN {X -3.966, Y 26.043, Z 96.900} C_DIS
   LIN {X -3.284, Y 22.918, Z 96.900} C_DIS
   LIN {X -2.257, Y 16.756, Z 96.900} C_DIS
   LIN {X -1.691, Y 10.737, Z 96.900}
   LaserEnd_Ext()
   LIN {X -6.719, Y 45.522, Z 96.900}
   LaserStart_Ext()
   LIN {X -5.229, Y 45.522, Z 96.900}
   LaserEnd_Ext()
   LIN {X -3.758, Y 44.522, Z 96.900}
   LaserStart_Ext()
   LIN {X -8.342, Y 44.522, Z 96.900}
   LaserEnd_Ext()
   LIN {X -8.881, Y 43.522, Z 96.900}
   LaserStart_Ext()
   LIN {X -3.070, Y 43.522, Z 96.900}
   LaserEnd_Ext()
   LIN {X -2.512, Y 42.522, Z 96.900}
   LaserStart_Ext()
   LIN {X -8.982, Y 42.522, Z 96.900}
   LaserEnd_Ext()
   LIN {X -8.728, Y 41.522, Z 96.900}
   LaserStart_Ext()
   LIN {X -1.960, Y 41.522, Z 96.900}
   LaserEnd_Ext()
   LIN {X -1.426, Y 40.522, Z 96.900}
   LaserStart_Ext()
   LIN {X -8.285, Y 40.522, Z 96.900}
   LaserEnd_Ext()
   LIN {X -7.807, Y 39.522, Z 96.900}
   LaserStart_Ext()
   LIN {X -0.906, Y 39.522, Z 96.900}
   LaserEnd_Ext()
   LIN {X -0.386, Y 38.522, Z 96.900}
   LaserStart_Ext()
   LIN {X -7.340, Y 38.522, Z 96.900}
   LaserEnd_Ext()
   LIN {X -6.899, Y 37.522, Z 96.900}
   LaserStart_Ext()
   LIN {X 0.082, Y 37.522, Z 96.900}
   LaserEnd_Ext()
   LIN {X 0.542, Y 36.522, Z 96.900}
   LaserStart_Ext()
   LIN {X -6.459, Y 36.522, Z 96.900}
   LaserEnd_Ext()
   LIN {X -6.085, Y 35.522, Z 96.900}
   LaserStart_Ext()
   LIN {X 1.001, Y 35.522, Z 96.900}
   LaserEnd_Ext()
   LIN {X 1.461, Y 34.522, Z 96.900}
   LaserStart_Ext()
   LIN {X -5.711, Y 34.522, Z 96.900}
   LaserEnd_Ext()
   LIN {X -5.337, Y 33.522, Z 96.900}
   LaserStart_Ext()
   LIN {X 1.921, Y 33.522, Z 96.900}
   LaserEnd_Ext()
   LIN {X 2.381, Y 32.522, Z 96.900}
   LaserStart_Ext()
   LIN {X -4.963, Y 32.522, Z 96.900}
   LaserEnd_Ext()
   LIN {X -4.589, Y 31.522, Z 96.900}
   LaserStart_Ext()
   LIN {X 2.841, Y 31.522, Z 96.900}
   LaserEnd_Ext()
   LIN {X 3.232, Y 30.522, Z 96.900}
   LaserStart_Ext()
   LIN {X -4.232, Y 30.522, Z 96.900}
   LaserEnd_Ext()
   LIN {X -3.941, Y 29.522, Z 96.900}
   LaserStart_Ext()
   LIN {X 3.594, Y 29.522, Z 96.900}
   LaserEnd_Ext()
   LIN {X 3.967, Y 28.522, Z 96.900}
   LaserStart_Ext()
   LIN {X -3.649, Y 28.522, Z 96.900}
   LaserEnd_Ext()
   LIN {X -3.356, Y 27.522, Z 96.900}
   LaserStart_Ext()
   LIN {X 4.340, Y 27.522, Z 96.900}
   LaserEnd_Ext()
   LIN {X 4.712, Y 26.522, Z 96.900}
   LaserStart_Ext()
   LIN {X -3.064, Y 26.522, Z 96.900}
   LaserEnd_Ext()
   LIN {X -2.829, Y 25.522, Z 96.900}
   LaserStart_Ext()
   LIN {X 5.085, Y 25.522, Z 96.900}
   LaserEnd_Ext()
   LIN {X 5.458, Y 24.522, Z 96.900}
   LaserStart_Ext()
   LIN {X -2.611, Y 24.522, Z 96.900}
   LaserEnd_Ext()
   LIN {X -2.392, Y 23.522, Z 96.900}
   LaserStart_Ext()
   LIN {X 5.825, Y 23.522, Z 96.900}
   LaserEnd_Ext()
   LIN {X 6.153, Y 22.522, Z 96.900}
   LaserStart_Ext()
   LIN {X -2.204, Y 22.522, Z 96.900}
   LaserEnd_Ext()
   LIN {X -2.038, Y 21.522, Z 96.900}
   LaserStart_Ext()
   LIN {X 6.481, Y 21.522, Z 96.900}
   LaserEnd_Ext()
   LIN {X 6.809, Y 20.522, Z 96.900}
   LaserStart_Ext()
   LIN {X -1.871, Y 20.522, Z 96.900}
   LaserEnd_Ext()
   LIN {X -1.704, Y 19.522, Z 96.900}
   LaserStart_Ext()
   LIN {X 7.072, Y 19.522, Z 96.900}
   LaserEnd_Ext()
   LIN {X 7.325, Y 18.522, Z 96.900}
   LaserStart_Ext()
   LIN {X -1.537, Y 18.522, Z 96.900}
   LaserEnd_Ext()
   LIN {X -1.371, Y 17.522, Z 96.900}
   LaserStart_Ext()
   LIN {X 7.578, Y 17.522, Z 96.900}
   LaserEnd_Ext()
   LIN {X 7.832, Y 16.522, Z 96.900}
   LaserStart_Ext()
   LIN {X -1.230, Y 16.522, Z 96.900}
   LaserEnd_Ext()
   LIN {X -1.136, Y 15.522, Z 96.900}
   LaserStart_Ext()
   LIN {X 8.085, Y 15.522, Z 96.900}
   LaserEnd_Ext()
   LIN {X 8.338, Y 14.522, Z 96.900}
   LaserStart_Ext()
   LIN {X -1.042, Y 14.522, Z 96.900}
   LaserEnd_Ext()
   LIN {X -0.948, Y 13.522, Z 96.900}
   LaserStart_Ext()
   LIN {X 8.591, Y 13.522, Z 96.900}
   LaserEnd_Ext()
   LIN {X 8.842, Y 12.522, Z 96.900}
   LaserStart_Ext()
   LIN {X -0.854, Y 12.522, Z 96.900}
   LaserEnd_Ext()
   LIN {X -0.760, Y 11.522, Z 96.900}
   LaserStart_Ext()
   LIN {X 9.093, Y 11.522, Z 96.900}
   LaserEnd_Ext()
   LIN {X 9.270, Y 10.522, Z 96.900}
   LaserStart_Ext()
   LIN {X -0.690, Y 10.522, Z 96.900}
   LaserEnd_Ext()
   LIN {X -0.686, Y 9.522, Z 96.900}
   LaserStart_Ext()
   LIN {X 9.433, Y 9.522, Z 96.900}
   LaserEnd_Ext()
   LIN {X 9.596, Y 8.522, Z 96.900}
   LaserStart_Ext()
   LIN {X -0.682, Y 8.522, Z 96.900}
   LaserEnd_Ext()
   LIN {X -0.678, Y 7.522, Z 96.900}
   LaserStart_Ext()
   LIN {X 9.760, Y 7.522, Z 96.900}
   LaserEnd_Ext()
   LIN {X 9.923, Y 6.522, Z 96.900}
   LaserStart_Ext()
   LIN {X -0.700, Y 6.522, Z 96.900}
   LaserEnd_Ext()
   LIN {X -0.737, Y 5.522, Z 96.900}
   LaserStart_Ext()
   LIN {X 10.086, Y 5.522, Z 96.900}
   LaserEnd_Ext()
   LIN {X 10.250, Y 4.522, Z 96.900}
   LaserStart_Ext()
   LIN {X -0.774, Y 4.522, Z 96.900}
   LaserEnd_Ext()
   LIN {X -0.811, Y 3.522, Z 96.900}
   LaserStart_Ext()
   LIN {X 10.413, Y 3.522, Z 96.900}
   LaserEnd_Ext()
   LIN {X 10.576, Y 2.522, Z 96.900}
   LaserStart_Ext()
   LIN {X -0.848, Y 2.522, Z 96.900}
   LaserEnd_Ext()
   LIN {X -0.897, Y 1.522, Z 96.900}
   LaserStart_Ext()
   LIN {X 10.715, Y 1.522, Z 96.900}
   LaserEnd_Ext()
   LIN {X 10.814, Y 0.522, Z 96.900}
   LaserStart_Ext()
   LIN {X -0.990, Y 0.522, Z 96.900}
   LaserEnd_Ext()
   LIN {X -1.092, Y -0.478, Z 96.900}
   LaserStart_Ext()
   LIN {X 10.913, Y -0.478, Z 96.900}
   LaserEnd_Ext()
   LIN {X 11.003, Y -1.478, Z 96.900}
   LaserStart_Ext()
   LIN {X -1.211, Y -1.478, Z 96.900}
   LaserEnd_Ext()
   LIN {X -1.346, Y -2.478, Z 96.900}
   LaserStart_Ext()
   LIN {X 11.084, Y -2.478, Z 96.900}
   LaserEnd_Ext()
   LIN {X 11.165, Y -3.478, Z 96.900}
   LaserStart_Ext()
   LIN {X -1.518, Y -3.478, Z 96.900}
   LaserEnd_Ext()
   LIN {X -1.690, Y -4.478, Z 96.900}
   LaserStart_Ext()
   LIN {X 11.226, Y -4.478, Z 96.900}
   LaserEnd_Ext()
   LIN {X 11.274, Y -5.478, Z 96.900}
   LaserStart_Ext()
   LIN {X -1.863, Y -5.478, Z 96.900}
   LaserEnd_Ext()
   LIN {X -2.035, Y -6.478, Z 96.900}
   LaserStart_Ext()
   LIN {X 11.317, Y -6.478, Z 96.900}
   LaserEnd_Ext()
   LIN {X 11.356, Y -7.478, Z 96.900}
   LaserStart_Ext()
   LIN {X -2.223, Y -7.478, Z 96.900}
   LaserEnd_Ext()
   LIN {X -2.446, Y -8.478, Z 96.900}
   LaserStart_Ext()
   LIN {X 11.395, Y -8.478, Z 96.900}
   LaserEnd_Ext()
   LIN {X 11.409, Y -9.478, Z 96.900}
   LaserStart_Ext()
   LIN {X -2.697, Y -9.478, Z 96.900}
   LaserEnd_Ext()
   LIN {X -2.948, Y -10.478, Z 96.900}
   LaserStart_Ext()
   LIN {X 11.414, Y -10.478, Z 96.900}
   LaserEnd_Ext()
   LIN {X 11.418, Y -11.478, Z 96.900}
   LaserStart_Ext()
   LIN {X -3.200, Y -11.478, Z 96.900}
   LaserEnd_Ext()
   LIN {X -3.457, Y -12.478, Z 96.900}
   LaserStart_Ext()
   LIN {X 1.443, Y -12.478, Z 96.900}
   LaserEnd_Ext()
   LIN {X 4.956, Y -12.478, Z 96.900}
   LaserStart_Ext()
   LIN {X 11.417, Y -12.478, Z 96.900}
   LaserEnd_Ext()
   LIN {X 11.388, Y -13.478, Z 96.900}
   LaserStart_Ext()
   LIN {X 6.931, Y -13.478, Z 96.900}
   LaserEnd_Ext()
   LIN {X -0.539, Y -13.478, Z 96.900}
   LaserStart_Ext()
   LIN {X -3.760, Y -13.478, Z 96.900}
   LaserEnd_Ext()
   LIN {X -4.072, Y -14.478, Z 96.900}
   LaserStart_Ext()
   LIN {X -1.443, Y -14.478, Z 96.900}
   LaserEnd_Ext()
   LIN {X 7.713, Y -14.478, Z 96.900}
   LaserStart_Ext()
   LIN {X 11.361, Y -14.478, Z 96.900}
   LaserEnd_Ext()
   LIN {X 11.334, Y -15.478, Z 96.900}
   LaserStart_Ext()
   LIN {X 8.491, Y -15.478, Z 96.900}
   LaserEnd_Ext()
   LIN {X -2.143, Y -15.478, Z 96.900}
   LaserStart_Ext()
   LIN {X -4.383, Y -15.478, Z 96.900}
   LaserEnd_Ext()
   LIN {X -4.545, Y -16.478, Z 96.900}
   LaserStart_Ext()
   LIN {X -2.371, Y -16.478, Z 96.900}
   LaserEnd_Ext()
   LIN {X 8.841, Y -16.478, Z 96.900}
   LaserStart_Ext()
   LIN {X 11.282, Y -16.478, Z 96.900}
   LaserEnd_Ext()
   LIN {X 11.225, Y -17.478, Z 96.900}
   LaserStart_Ext()
   LIN {X 9.018, Y -17.478, Z 96.900}
   LaserEnd_Ext()
   LIN {X -2.599, Y -17.478, Z 96.900}
   LaserStart_Ext()
   LIN {X -4.691, Y -17.478, Z 96.900}
   LaserEnd_Ext()
   LIN {X -4.829, Y -18.478, Z 96.900}
   LaserStart_Ext()
   LIN {X -2.822, Y -18.478, Z 96.900}
   LaserEnd_Ext()
   LIN {X 9.150, Y -18.478, Z 96.900}
   LaserStart_Ext()
   LIN {X 11.167, Y -18.478, Z 96.900}
   LaserEnd_Ext()
   LIN {X 10.947, Y -19.478, Z 96.900}
   LaserStart_Ext()
   LIN {X 8.872, Y -19.478, Z 96.900}
   LaserEnd_Ext()
   LIN {X -2.617, Y -19.478, Z 96.900}
   LaserStart_Ext()
   LIN {X -4.591, Y -19.478, Z 96.900}
   LaserEnd_Ext()
   LIN {X -4.349, Y -20.478, Z 96.900}
   LaserStart_Ext()
   LIN {X -2.316, Y -20.478, Z 96.900}
   LaserEnd_Ext()
   LIN {X 8.580, Y -20.478, Z 96.900}
   LaserStart_Ext()
   LIN {X 10.707, Y -20.478, Z 96.900}
   LaserEnd_Ext()
   LIN {X 10.330, Y -21.478, Z 96.900}
   LaserStart_Ext()
   LIN {X 8.072, Y -21.478, Z 96.900}
   LaserEnd_Ext()
   LIN {X -1.802, Y -21.478, Z 96.900}
   LaserStart_Ext()
   LIN {X -4.106, Y -21.478, Z 96.900}
   LaserEnd_Ext()
   LIN {X -3.495, Y -22.478, Z 96.900}
   LaserStart_Ext()
   LIN {X -0.927, Y -22.478, Z 96.900}
   LaserEnd_Ext()
   LIN {X 7.170, Y -22.478, Z 96.900}
   LaserStart_Ext()
   LIN {X 9.617, Y -22.478, Z 96.900}
   LaserEnd_Ext()
   LIN {X 8.905, Y -23.478, Z 96.900}
   LaserStart_Ext()
   LIN {X 5.677, Y -23.478, Z 96.900}
   LaserEnd_Ext()
   LIN {X 0.563, Y -23.478, Z 96.900}
   LaserStart_Ext()
   LIN {X -2.796, Y -23.478, Z 96.900}
   LaserEnd_Ext()
   LIN {X -1.521, Y -24.478, Z 96.900}
   LaserStart_Ext()
   LIN {X 7.848, Y -24.478, Z 96.900}
   LaserEnd_Ext()
   LIN {X 6.102, Y -25.478, Z 96.900}
   LaserStart_Ext()
   LIN {X 0.011, Y -25.478, Z 96.900}
   LaserEnd_Ext()
   LIN {X 0.317, Y -14.054, Z 97.750}
   LaserStart_Ext()
   LIN {X 1.997, Y -13.302, Z 97.750} C_DIS
   LIN {X 2.193, Y -13.214, Z 97.750} C_DIS
   LIN {X 4.360, Y -13.210, Z 97.750} C_DIS
   LIN {X 6.057, Y -14.003, Z 97.750} C_DIS
   LIN {X 6.286, Y -14.109, Z 97.750} C_DIS
   LIN {X 6.497, Y -14.378, Z 97.750} C_DIS
   LIN {X 7.849, Y -16.114, Z 97.750} C_DIS
   LIN {X 8.202, Y -18.077, Z 97.750} C_DIS
   LIN {X 8.240, Y -18.289, Z 97.750} C_DIS
   LIN {X 8.151, Y -18.597, Z 97.750} C_DIS
   LIN {X 7.581, Y -20.560, Z 97.750} C_DIS
   LIN {X 6.407, Y -21.863, Z 97.750} C_DIS
   LIN {X 6.130, Y -22.173, Z 97.750} C_DIS
   LIN {X 5.893, Y -22.279, Z 97.750} C_DIS
   LIN {X 4.194, Y -23.010, Z 97.750} C_DIS
   LIN {X 2.487, Y -22.999, Z 97.750} C_DIS
   LIN {X 2.107, Y -22.994, Z 97.750} C_DIS
   LIN {X 1.630, Y -22.773, Z 97.750} C_DIS
   LIN {X 0.230, Y -22.127, Z 97.750} C_DIS
   LIN {X -0.541, Y -21.253, Z 97.750} C_DIS
   LIN {X -1.145, Y -20.563, Z 97.750} C_DIS
   LIN {X -1.431, Y -19.611, Z 97.750} C_DIS
   LIN {X -1.749, Y -18.566, Z 97.750} C_DIS
   LIN {X -1.386, Y -16.966, Z 97.750} C_DIS
   LIN {X -1.072, Y -15.590, Z 97.750} C_DIS
   LIN {X -0.553, Y -15.015, Z 97.750} C_DIS
   LIN {X 0.317, Y -14.054, Z 97.750}
   LaserEnd_Ext()
   LIN {X 3.617, Y 32.172, Z 97.750}
   LaserStart_Ext()
   LIN {X 0.553, Y 38.839, Z 97.750} C_DIS
   LIN {X -0.382, Y 40.636, Z 97.750} C_DIS
   LIN {X -0.989, Y 41.776, Z 97.750} C_DIS
   LIN {X -1.273, Y 42.291, Z 97.750} C_DIS
   LIN {X -1.917, Y 43.451, Z 97.750} C_DIS
   LIN {X -2.608, Y 44.668, Z 97.750} C_DIS
   LIN {X -2.693, Y 44.791, Z 97.750} C_DIS
   LIN {X -3.617, Y 45.851, Z 97.750} C_DIS
   LIN {X -4.823, Y 46.444, Z 97.750} C_DIS
   LIN {X -5.179, Y 46.618, Z 97.750} C_DIS
   LIN {X -5.788, Y 46.627, Z 97.750} C_DIS
   LIN {X -6.924, Y 46.648, Z 97.750} C_DIS
   LIN {X -7.503, Y 46.290, Z 97.750} C_DIS
   LIN {X -9.221, Y 45.236, Z 97.750} C_DIS
   LIN {X -9.567, Y 44.548, Z 97.750} C_DIS
   LIN {X -9.959, Y 43.775, Z 97.750} C_DIS
   LIN {X -10.019, Y 42.995, Z 97.750} C_DIS
   LIN {X -10.067, Y 42.318, Z 97.750} C_DIS
   LIN {X -9.870, Y 41.686, Z 97.750} C_DIS
   LIN {X -9.637, Y 40.933, Z 97.750} C_DIS
   LIN {X -9.428, Y 40.506, Z 97.750} C_DIS
   LIN {X -9.089, Y 39.809, Z 97.750} C_DIS
   LIN {X -8.438, Y 38.443, Z 97.750} C_DIS
   LIN {X -8.365, Y 38.285, Z 97.750} C_DIS
   LIN {X -7.446, Y 36.217, Z 97.750} C_DIS
   LIN {X -7.308, Y 35.893, Z 97.750} C_DIS
   LIN {X -5.402, Y 30.786, Z 97.750} C_DIS
   LIN {X -5.123, Y 29.974, Z 97.750} C_DIS
   LIN {X -4.009, Y 26.161, Z 97.750} C_DIS
   LIN {X -3.094, Y 21.969, Z 97.750} C_DIS
   LIN {X -2.307, Y 17.252, Z 97.750} C_DIS
   LIN {X -1.661, Y 10.378, Z 97.750} C_DIS
   LIN {X -1.650, Y 7.524, Z 97.750} C_DIS
   LIN {X -1.875, Y 1.428, Z 97.750} C_DIS
   LIN {X -2.012, Y -0.038, Z 97.750} C_DIS
   LIN {X -2.059, Y -0.412, Z 97.750} C_DIS
   LIN {X -2.212, Y -1.716, Z 97.750} C_DIS
   LIN {X -2.334, Y -2.531, Z 97.750} C_DIS
   LIN {X -3.198, Y -7.520, Z 97.750} C_DIS
   LIN {X -3.248, Y -7.725, Z 97.750} C_DIS
   LIN {X -4.417, Y -12.409, Z 97.750} C_DIS
   LIN {X -4.641, Y -13.143, Z 97.750} C_DIS
   LIN {X -5.317, Y -15.312, Z 97.750} C_DIS
   LIN {X -5.719, Y -18.068, Z 97.750} C_DIS
   LIN {X -5.773, Y -18.451, Z 97.750} C_DIS
   LIN {X -5.666, Y -18.881, Z 97.750} C_DIS
   LIN {X -4.895, Y -22.055, Z 97.750} C_DIS
   LIN {X -3.487, Y -24.062, Z 97.750} C_DIS
   LIN {X -3.206, Y -24.459, Z 97.750} C_DIS
   LIN {X -2.653, Y -24.816, Z 97.750} C_DIS
   LIN {X -0.012, Y -26.540, Z 97.750} C_DIS
   LIN {X 2.122, Y -26.929, Z 97.750} C_DIS
   LIN {X 3.896, Y -27.018, Z 97.750} C_DIS
   LIN {X 6.194, Y -26.600, Z 97.750} C_DIS
   LIN {X 6.927, Y -26.190, Z 97.750} C_DIS
   LIN {X 9.281, Y -24.752, Z 97.750} C_DIS
   LIN {X 10.703, Y -22.756, Z 97.750} C_DIS
   LIN {X 11.553, Y -21.533, Z 97.750} C_DIS
   LIN {X 11.964, Y -19.787, Z 97.750} C_DIS
   LIN {X 12.236, Y -18.651, Z 97.750} C_DIS
   LIN {X 12.281, Y -17.874, Z 97.750} C_DIS
   LIN {X 12.410, Y -15.394, Z 97.750} C_DIS
   LIN {X 12.477, Y -12.823, Z 97.750} C_DIS
   LIN {X 12.485, Y -12.436, Z 97.750} C_DIS
   LIN {X 12.477, Y -11.268, Z 97.750} C_DIS
   LIN {X 12.464, Y -8.631, Z 97.750} C_DIS
   LIN {X 12.419, Y -7.483, Z 97.750} C_DIS
   LIN {X 12.236, Y -3.635, Z 97.750} C_DIS
   LIN {X 12.065, Y -1.523, Z 97.750} C_DIS
   LIN {X 11.721, Y 1.964, Z 97.750} C_DIS
   LIN {X 10.617, Y 8.726, Z 97.750} C_DIS
   LIN {X 10.190, Y 11.332, Z 97.750} C_DIS
   LIN {X 9.375, Y 14.584, Z 97.750} C_DIS
   LIN {X 7.895, Y 20.432, Z 97.750} C_DIS
   LIN {X 6.620, Y 24.319, Z 97.750} C_DIS
   LIN {X 4.113, Y 31.044, Z 97.750} C_DIS
   LIN {X 3.932, Y 31.499, Z 97.750} C_DIS
   LIN {X 3.826, Y 31.722, Z 97.750} C_DIS
   LIN {X 3.617, Y 32.172, Z 97.750}
   LaserEnd_Ext()
   LIN {X -8.280, Y 44.640, Z 97.750}
   LaserStart_Ext()
   LIN {X -8.280, Y 40.432, Z 97.750}
   LaserEnd_Ext()
   LIN {X -7.280, Y 38.307, Z 97.750}
   LaserStart_Ext()
   LIN {X -7.280, Y 45.254, Z 97.750}
   LaserEnd_Ext()
   LIN {X -6.280, Y 45.636, Z 97.750}
   LaserStart_Ext()
   LIN {X -6.280, Y 35.998, Z 97.750}
   LaserEnd_Ext()
   LIN {X -5.280, Y 33.319, Z 97.750}
   LaserStart_Ext()
   LIN {X -5.280, Y 45.554, Z 97.750}
   LaserEnd_Ext()
   LIN {X -4.280, Y 45.062, Z 97.750}
   LaserStart_Ext()
   LIN {X -4.280, Y 30.598, Z 97.750}
   LaserEnd_Ext()
   LIN {X -4.280, Y -15.345, Z 97.750}
   LaserStart_Ext()
   LIN {X -4.280, Y -20.352, Z 97.750}
   LaserEnd_Ext()
   LIN {X -3.280, Y -22.617, Z 97.750}
   LaserStart_Ext()
   LIN {X -3.280, Y -11.984, Z 97.750}
   LaserEnd_Ext()
   LIN {X -3.280, Y 27.233, Z 97.750}
   LaserStart_Ext()
   LIN {X -3.280, Y 43.825, Z 97.750}
   LaserEnd_Ext()
   LIN {X -2.280, Y 42.044, Z 97.750}
   LaserStart_Ext()
   LIN {X -2.280, Y 22.930, Z 97.750}
   LaserEnd_Ext()
   LIN {X -2.280, Y -7.976, Z 97.750}
   LaserStart_Ext()
   LIN {X -2.280, Y -16.388, Z 97.750}
   LaserEnd_Ext()
   LIN {X -2.280, Y -20.261, Z 97.750}
   LaserStart_Ext()
   LIN {X -2.280, Y -23.867, Z 97.750}
   LaserEnd_Ext()
   LIN {X -1.280, Y -24.518, Z 97.750}
   LaserStart_Ext()
   LIN {X -1.280, Y -21.927, Z 97.750}
   LaserEnd_Ext()
   LIN {X -1.280, Y -14.328, Z 97.750}
   LaserStart_Ext()
   LIN {X -1.280, Y -2.242, Z 97.750}
   LaserEnd_Ext()
   LIN {X -1.280, Y 17.008, Z 97.750}
   LaserStart_Ext()
   LIN {X -1.280, Y 40.195, Z 97.750}
   LaserEnd_Ext()
   LIN {X -0.280, Y 38.256, Z 97.750}
   LaserStart_Ext()
   LIN {X -0.280, Y -13.252, Z 97.750}
   LaserEnd_Ext()
   LIN {X -0.280, Y -22.987, Z 97.750}
   LaserStart_Ext()
   LIN {X -0.280, Y -25.171, Z 97.750}
   LaserEnd_Ext()
   LIN {X 0.720, Y -25.657, Z 97.750}
   LaserStart_Ext()
   LIN {X 0.720, Y -23.454, Z 97.750}
   LaserEnd_Ext()
   LIN {X 0.720, Y -12.778, Z 97.750}
   LaserStart_Ext()
   LIN {X 0.720, Y 36.080, Z 97.750}
   LaserEnd_Ext()
   LIN {X 1.720, Y 33.904, Z 97.750}
   LaserStart_Ext()
   LIN {X 1.720, Y -12.330, Z 97.750}
   LaserEnd_Ext()
   LIN {X 1.720, Y -23.915, Z 97.750}
   LaserStart_Ext()
   LIN {X 1.720, Y -25.839, Z 97.750}
   LaserEnd_Ext()
   LIN {X 2.720, Y -25.957, Z 97.750}
   LaserStart_Ext()
   LIN {X 2.720, Y -24.001, Z 97.750}
   LaserEnd_Ext()
   LIN {X 2.720, Y -12.214, Z 97.750}
   LaserStart_Ext()
   LIN {X 2.720, Y 31.729, Z 97.750}
   LaserEnd_Ext()
   LIN {X 3.720, Y 29.235, Z 97.750}
   LaserStart_Ext()
   LIN {X 3.720, Y -12.211, Z 97.750}
   LaserEnd_Ext()
   LIN {X 3.720, Y -24.007, Z 97.750}
   LaserStart_Ext()
   LIN {X 3.720, Y -26.008, Z 97.750}
   LaserEnd_Ext()
   LIN {X 4.720, Y -25.852, Z 97.750}
   LaserStart_Ext()
   LIN {X 4.720, Y -23.872, Z 97.750}
   LaserEnd_Ext()
   LIN {X 4.720, Y -12.279, Z 97.750}
   LaserStart_Ext()
   LIN {X 4.720, Y 26.552, Z 97.750}
   LaserEnd_Ext()
   LIN {X 5.720, Y 23.853, Z 97.750}
   LaserStart_Ext()
   LIN {X 5.720, Y -12.742, Z 97.750}
   LaserEnd_Ext()
   LIN {X 5.720, Y -23.442, Z 97.750}
   LaserStart_Ext()
   LIN {X 5.720, Y -25.670, Z 97.750}
   LaserEnd_Ext()
   LIN {X 6.720, Y -25.144, Z 97.750}
   LaserStart_Ext()
   LIN {X 6.720, Y -22.980, Z 97.750}
   LaserEnd_Ext()
   LIN {X 6.720, Y -13.209, Z 97.750}
   LaserStart_Ext()
   LIN {X 6.720, Y 20.805, Z 97.750}
   LaserEnd_Ext()
   LIN {X 7.720, Y 17.048, Z 97.750}
   LaserStart_Ext()
   LIN {X 7.720, Y -14.321, Z 97.750}
   LaserEnd_Ext()
   LIN {X 7.720, Y -21.899, Z 97.750}
   LaserStart_Ext()
   LIN {X 7.720, Y -24.534, Z 97.750}
   LaserEnd_Ext()
   LIN {X 8.720, Y -23.817, Z 97.750}
   LaserStart_Ext()
   LIN {X 8.720, Y -20.223, Z 97.750}
   LaserEnd_Ext()
   LIN {X 8.720, Y -15.625, Z 97.750}
   LaserStart_Ext()
   LIN {X 8.720, Y 13.085, Z 97.750}
   LaserEnd_Ext()
   LIN {X 9.720, Y 8.011, Z 97.750}
   LaserStart_Ext()
   LIN {X 9.720, Y -22.413, Z 97.750}
   LaserEnd_Ext()
   LIN {X 10.720, Y -20.706, Z 97.750}
   LaserStart_Ext()
   LIN {X 10.720, Y 1.887, Z 97.750}
   LaserEnd_Ext()
   LIN {X -1.666, Y -18.519, Z 98.600}
   LaserStart_Ext()
   LIN {X -1.152, Y -16.253, Z 98.600} C_DIS
   LIN {X -0.987, Y -15.526, Z 98.600} C_DIS
   LIN {X -0.591, Y -15.088, Z 98.600} C_DIS
   LIN {X 0.397, Y -13.996, Z 98.600} C_DIS
   LIN {X 1.325, Y -13.581, Z 98.600} C_DIS
   LIN {X 2.270, Y -13.157, Z 98.600} C_DIS
   LIN {X 3.741, Y -13.150, Z 98.600} C_DIS
   LIN {X 4.430, Y -13.149, Z 98.600} C_DIS
   LIN {X 4.920, Y -13.378, Z 98.600} C_DIS
   LIN {X 6.358, Y -14.043, Z 98.600} C_DIS
   LIN {X 7.682, Y -15.731, Z 98.600} C_DIS
   LIN {X 7.926, Y -16.044, Z 98.600} C_DIS
   LIN {X 7.990, Y -16.399, Z 98.600} C_DIS
   LIN {X 8.322, Y -18.218, Z 98.600} C_DIS
   LIN {X 7.720, Y -20.304, Z 98.600} C_DIS
   LIN {X 7.667, Y -20.493, Z 98.600} C_DIS
   LIN {X 7.538, Y -20.642, Z 98.600} C_DIS
   LIN {X 6.245, Y -22.090, Z 98.600} C_DIS
   LIN {X 4.842, Y -22.717, Z 98.600} C_DIS
   LIN {X 4.316, Y -22.943, Z 98.600} C_DIS
   LIN {X 3.499, Y -22.938, Z 98.600} C_DIS
   LIN {X 2.200, Y -22.938, Z 98.600} C_DIS
   LIN {X 1.406, Y -22.576, Z 98.600} C_DIS
   LIN {X 0.322, Y -22.076, Z 98.600} C_DIS
   LIN {X -0.719, Y -20.896, Z 98.600} C_DIS
   LIN {X -1.057, Y -20.515, Z 98.600} C_DIS
   LIN {X -1.195, Y -20.069, Z 98.600} C_DIS
   LIN {X -1.666, Y -18.519, Z 98.600}
   LaserEnd_Ext()
   LIN {X -9.885, Y 41.586, Z 98.600}
   LaserStart_Ext()
   LIN {X -9.692, Y 40.962, Z 98.600} C_DIS
   LIN {X -9.330, Y 40.223, Z 98.600} C_DIS
   LIN {X -9.141, Y 39.839, Z 98.600} C_DIS
   LIN {X -8.941, Y 39.422, Z 98.600} C_DIS
   LIN {X -8.449, Y 38.397, Z 98.600} C_DIS
   LIN {X -7.574, Y 36.440, Z 98.600} C_DIS
   LIN {X -7.498, Y 36.269, Z 98.600} C_DIS
   LIN {X -7.220, Y 35.616, Z 98.600} C_DIS
   LIN {X -5.605, Y 31.288, Z 98.600} C_DIS
   LIN {X -5.003, Y 29.538, Z 98.600} C_DIS
   LIN {X -4.051, Y 26.279, Z 98.600} C_DIS
   LIN {X -2.903, Y 21.020, Z 98.600} C_DIS
   LIN {X -2.357, Y 17.748, Z 98.600} C_DIS
   LIN {X -1.630, Y 10.018, Z 98.600} C_DIS
   LIN {X -1.622, Y 7.875, Z 98.600} C_DIS
   LIN {X -1.874, Y 1.069, Z 98.600} C_DIS
   LIN {X -1.971, Y 0.026, Z 98.600} C_DIS
   LIN {X -2.005, Y -0.240, Z 98.600} C_DIS
   LIN {X -2.114, Y -1.169, Z 98.600} C_DIS
   LIN {X -2.506, Y -3.801, Z 98.600} C_DIS
   LIN {X -3.147, Y -7.501, Z 98.600} C_DIS
   LIN {X -3.529, Y -9.077, Z 98.600} C_DIS
   LIN {X -4.356, Y -12.392, Z 98.600} C_DIS
   LIN {X -4.958, Y -14.358, Z 98.600} C_DIS
   LIN {X -5.243, Y -15.274, Z 98.600} C_DIS
   LIN {X -5.413, Y -16.437, Z 98.600} C_DIS
   LIN {X -5.692, Y -18.413, Z 98.600} C_DIS
   LIN {X -5.141, Y -20.635, Z 98.600} C_DIS
   LIN {X -4.805, Y -22.016, Z 98.600} C_DIS
   LIN {X -4.192, Y -22.889, Z 98.600} C_DIS
   LIN {X -3.111, Y -24.415, Z 98.600} C_DIS
   LIN {X -0.986, Y -25.786, Z 98.600} C_DIS
   LIN {X 0.093, Y -26.490, Z 98.600} C_DIS
   LIN {X 3.077, Y -27.034, Z 98.600} C_DIS
   LIN {X 3.352, Y -27.048, Z 98.600} C_DIS
   LIN {X 4.208, Y -26.893, Z 98.600} C_DIS
   LIN {X 6.444, Y -26.481, Z 98.600} C_DIS
   LIN {X 7.647, Y -25.727, Z 98.600} C_DIS
   LIN {X 9.409, Y -24.652, Z 98.600} C_DIS
   LIN {X 9.930, Y -23.921, Z 98.600} C_DIS
   LIN {X 11.642, Y -21.455, Z 98.600} C_DIS
   LIN {X 12.219, Y -19.004, Z 98.600} C_DIS
   LIN {X 12.318, Y -18.572, Z 98.600} C_DIS
   LIN {X 12.359, Y -17.742, Z 98.600} C_DIS
   LIN {X 12.485, Y -15.314, Z 98.600} C_DIS
   LIN {X 12.519, Y -13.997, Z 98.600} C_DIS
   LIN {X 12.552, Y -12.355, Z 98.600} C_DIS
   LIN {X 12.528, Y -8.942, Z 98.600} C_DIS
   LIN {X 12.523, Y -8.551, Z 98.600} C_DIS
   LIN {X 12.482, Y -7.786, Z 98.600} C_DIS
   LIN {X 12.276, Y -3.458, Z 98.600} C_DIS
   LIN {X 12.166, Y -2.105, Z 98.600} C_DIS
   LIN {X 11.771, Y 1.904, Z 98.600} C_DIS
   LIN {X 10.871, Y 7.414, Z 98.600} C_DIS
   LIN {X 10.270, Y 11.093, Z 98.600} C_DIS
   LIN {X 9.119, Y 15.683, Z 98.600} C_DIS
   LIN {X 7.977, Y 20.194, Z 98.600} C_DIS
   LIN {X 6.511, Y 24.661, Z 98.600} C_DIS
   LIN {X 4.641, Y 29.679, Z 98.600} C_DIS
   LIN {X 3.852, Y 31.666, Z 98.600} C_DIS
   LIN {X 3.387, Y 32.640, Z 98.600} C_DIS
   LIN {X 2.474, Y 34.605, Z 98.600} C_DIS
   LIN {X 0.520, Y 38.856, Z 98.600} C_DIS
   LIN {X -0.076, Y 40.001, Z 98.600} C_DIS
   LIN {X -0.619, Y 41.021, Z 98.600} C_DIS
   LIN {X -1.045, Y 41.823, Z 98.600} C_DIS
   LIN {X -1.780, Y 43.141, Z 98.600} C_DIS
   LIN {X -1.978, Y 43.498, Z 98.600} C_DIS
   LIN {X -2.091, Y 43.696, Z 98.600} C_DIS
   LIN {X -2.714, Y 44.786, Z 98.600} C_DIS
   LIN {X -3.608, Y 45.808, Z 98.600} C_DIS
   LIN {X -3.684, Y 45.894, Z 98.600} C_DIS
   LIN {X -3.840, Y 45.970, Z 98.600} C_DIS
   LIN {X -5.247, Y 46.657, Z 98.600} C_DIS
   LIN {X -6.304, Y 46.674, Z 98.600} C_DIS
   LIN {X -6.992, Y 46.683, Z 98.600} C_DIS
   LIN {X -7.698, Y 46.246, Z 98.600} C_DIS
   LIN {X -9.279, Y 45.274, Z 98.600} C_DIS
   LIN {X -9.680, Y 44.493, Z 98.600} C_DIS
   LIN {X -10.009, Y 43.843, Z 98.600} C_DIS
   LIN {X -10.059, Y 43.196, Z 98.600} C_DIS
   LIN {X -10.117, Y 42.292, Z 98.600} C_DIS
   LIN {X -9.885, Y 41.586, Z 98.600}
   LaserEnd_Ext()
   LIN {X 0.190, Y -25.360, Z 98.600}
   LaserStart_Ext()
   LIN {X 6.350, Y -25.360, Z 98.600}
   LaserEnd_Ext()
   LIN {X 7.968, Y -24.360, Z 98.600}
   LaserStart_Ext()
   LIN {X -1.352, Y -24.360, Z 98.600}
   LaserEnd_Ext()
   LIN {X -2.633, Y -23.360, Z 98.600}
   LaserStart_Ext()
   LIN {X 0.719, Y -23.360, Z 98.600}
   LaserEnd_Ext()
   LIN {X 5.854, Y -23.360, Z 98.600}
   LaserStart_Ext()
   LIN {X 9.102, Y -23.360, Z 98.600}
   LaserEnd_Ext()
   LIN {X 9.796, Y -22.360, Z 98.600}
   LaserStart_Ext()
   LIN {X 7.345, Y -22.360, Z 98.600}
   LaserEnd_Ext()
   LIN {X -0.761, Y -22.360, Z 98.600}
   LaserStart_Ext()
   LIN {X -3.342, Y -22.360, Z 98.600}
   LaserEnd_Ext()
   LIN {X -3.935, Y -21.360, Z 98.600}
   LaserStart_Ext()
   LIN {X -1.644, Y -21.360, Z 98.600}
   LaserEnd_Ext()
   LIN {X 8.238, Y -21.360, Z 98.600}
   LaserStart_Ext()
   LIN {X 10.490, Y -21.360, Z 98.600}
   LaserEnd_Ext()
   LIN {X 10.872, Y -20.360, Z 98.600}
   LaserStart_Ext()
   LIN {X 8.745, Y -20.360, Z 98.600}
   LaserEnd_Ext()
   LIN {X -2.151, Y -20.360, Z 98.600}
   LaserStart_Ext()
   LIN {X -4.178, Y -20.360, Z 98.600}
   LaserEnd_Ext()
   LIN {X -4.426, Y -19.360, Z 98.600}
   LaserStart_Ext()
   LIN {X -2.456, Y -19.360, Z 98.600}
   LaserEnd_Ext()
   LIN {X 9.034, Y -19.360, Z 98.600}
   LaserStart_Ext()
   LIN {X 11.108, Y -19.360, Z 98.600}
   LaserEnd_Ext()
   LIN {X 11.327, Y -18.360, Z 98.600}
   LaserStart_Ext()
   LIN {X 9.311, Y -18.360, Z 98.600}
   LaserEnd_Ext()
   LIN {X -2.652, Y -18.360, Z 98.600}
   LaserStart_Ext()
   LIN {X -4.674, Y -18.360, Z 98.600}
   LaserEnd_Ext()
   LIN {X -4.533, Y -17.360, Z 98.600}
   LaserStart_Ext()
   LIN {X -2.429, Y -17.360, Z 98.600}
   LaserEnd_Ext()
   LIN {X 9.182, Y -17.360, Z 98.600}
   LaserStart_Ext()
   LIN {X 11.377, Y -17.360, Z 98.600}
   LaserEnd_Ext()
   LIN {X 11.429, Y -16.360, Z 98.600}
   LaserStart_Ext()
   LIN {X 8.999, Y -16.360, Z 98.600}
   LaserEnd_Ext()
   LIN {X -2.202, Y -16.360, Z 98.600}
   LaserStart_Ext()
   LIN {X -4.391, Y -16.360, Z 98.600}
   LaserEnd_Ext()
   LIN {X -4.223, Y -15.360, Z 98.600}
   LaserStart_Ext()
   LIN {X -1.975, Y -15.360, Z 98.600}
   LaserEnd_Ext()
   LIN {X 8.661, Y -15.360, Z 98.600}
   LaserStart_Ext()
   LIN {X 11.481, Y -15.360, Z 98.600}
   LaserEnd_Ext()
   LIN {X 11.509, Y -14.360, Z 98.600}
   LaserStart_Ext()
   LIN {X 7.878, Y -14.360, Z 98.600}
   LaserEnd_Ext()
   LIN {X -1.281, Y -14.360, Z 98.600}
   LaserStart_Ext()
   LIN {X -3.913, Y -14.360, Z 98.600}
   LaserEnd_Ext()
   LIN {X -3.607, Y -13.360, Z 98.600}
   LaserStart_Ext()
   LIN {X -0.376, Y -13.360, Z 98.600}
   LaserEnd_Ext()
   LIN {X 7.088, Y -13.360, Z 98.600}
   LaserStart_Ext()
   LIN {X 11.532, Y -13.360, Z 98.600}
   LaserEnd_Ext()
   LIN {X 11.552, Y -12.360, Z 98.600}
   LaserStart_Ext()
   LIN {X 5.104, Y -12.360, Z 98.600}
   LaserEnd_Ext()
   LIN {X 1.603, Y -12.360, Z 98.600}
   LaserStart_Ext()
   LIN {X -3.317, Y -12.360, Z 98.600}
   LaserEnd_Ext()
   LIN {X -3.068, Y -11.360, Z 98.600}
   LaserStart_Ext()
   LIN {X 11.545, Y -11.360, Z 98.600}
   LaserEnd_Ext()
   LIN {X 11.538, Y -10.360, Z 98.600}
   LaserStart_Ext()
   LIN {X -2.818, Y -10.360, Z 98.600}
   LaserEnd_Ext()
   LIN {X -2.569, Y -9.360, Z 98.600}
   LaserStart_Ext()
   LIN {X 11.531, Y -9.360, Z 98.600}
   LaserEnd_Ext()
   LIN {X 11.511, Y -8.360, Z 98.600}
   LaserStart_Ext()
   LIN {X -2.326, Y -8.360, Z 98.600}
   LaserEnd_Ext()
   LIN {X -2.108, Y -7.360, Z 98.600}
   LaserStart_Ext()
   LIN {X 11.461, Y -7.360, Z 98.600}
   LaserEnd_Ext()
   LIN {X 11.413, Y -6.360, Z 98.600}
   LaserStart_Ext()
   LIN {X -1.935, Y -6.360, Z 98.600}
   LaserEnd_Ext()
   LIN {X -1.762, Y -5.360, Z 98.600}
   LaserStart_Ext()
   LIN {X 11.365, Y -5.360, Z 98.600}
   LaserEnd_Ext()
   LIN {X 11.318, Y -4.360, Z 98.600}
   LaserStart_Ext()
   LIN {X -1.588, Y -4.360, Z 98.600}
   LaserEnd_Ext()
   LIN {X -1.430, Y -3.360, Z 98.600}
   LaserStart_Ext()
   LIN {X 11.265, Y -3.360, Z 98.600}
   LaserEnd_Ext()
   LIN {X 11.184, Y -2.360, Z 98.600}
   LaserStart_Ext()
   LIN {X -1.281, Y -2.360, Z 98.600}
   LaserEnd_Ext()
   LIN {X -1.132, Y -1.360, Z 98.600}
   LaserStart_Ext()
   LIN {X 11.088, Y -1.360, Z 98.600}
   LaserEnd_Ext()
   LIN {X 10.989, Y -0.360, Z 98.600}
   LaserStart_Ext()
   LIN {X -1.012, Y -0.360, Z 98.600}
   LaserEnd_Ext()
   LIN {X -0.910, Y 0.640, Z 98.600}
   LaserStart_Ext()
   LIN {X 10.891, Y 0.640, Z 98.600}
   LaserEnd_Ext()
   LIN {X 10.792, Y 1.640, Z 98.600}
   LaserStart_Ext()
   LIN {X -0.852, Y 1.640, Z 98.600}
   LaserEnd_Ext()
   LIN {X -0.815, Y 2.640, Z 98.600}
   LaserStart_Ext()
   LIN {X 10.637, Y 2.640, Z 98.600}
   LaserEnd_Ext()
   LIN {X 10.474, Y 3.640, Z 98.600}
   LaserStart_Ext()
   LIN {X -0.778, Y 3.640, Z 98.600}
   LaserEnd_Ext()
   LIN {X -0.741, Y 4.640, Z 98.600}
   LaserStart_Ext()
   LIN {X 10.311, Y 4.640, Z 98.600}
   LaserEnd_Ext()
   LIN {X 10.148, Y 5.640, Z 98.600}
   LaserStart_Ext()
   LIN {X -0.704, Y 5.640, Z 98.600}
   LaserEnd_Ext()
   LIN {X -0.667, Y 6.640, Z 98.600}
   LaserStart_Ext()
   LIN {X 9.984, Y 6.640, Z 98.600}
   LaserEnd_Ext()
   LIN {X 9.821, Y 7.640, Z 98.600}
   LaserStart_Ext()
   LIN {X -0.630, Y 7.640, Z 98.600}
   LaserEnd_Ext()
   LIN {X -0.625, Y 8.640, Z 98.600}
   LaserStart_Ext()
   LIN {X 9.657, Y 8.640, Z 98.600}
   LaserEnd_Ext()
   LIN {X 9.494, Y 9.640, Z 98.600}
   LaserStart_Ext()
   LIN {X -0.629, Y 9.640, Z 98.600}
   LaserEnd_Ext()
   LIN {X -0.684, Y 10.640, Z 98.600}
   LaserStart_Ext()
   LIN {X 9.330, Y 10.640, Z 98.600}
   LaserEnd_Ext()
   LIN {X 9.101, Y 11.640, Z 98.600}
   LaserStart_Ext()
   LIN {X -0.779, Y 11.640, Z 98.600}
   LaserEnd_Ext()
   LIN {X -0.873, Y 12.640, Z 98.600}
   LaserStart_Ext()
   LIN {X 8.851, Y 12.640, Z 98.600}
   LaserEnd_Ext()
   LIN {X 8.600, Y 13.640, Z 98.600}
   LaserStart_Ext()
   LIN {X -0.967, Y 13.640, Z 98.600}
   LaserEnd_Ext()
   LIN {X -1.061, Y 14.640, Z 98.600}
   LaserStart_Ext()
   LIN {X 8.349, Y 14.640, Z 98.600}
   LaserEnd_Ext()
   LIN {X 8.098, Y 15.640, Z 98.600}
   LaserStart_Ext()
   LIN {X -1.155, Y 15.640, Z 98.600}
   LaserEnd_Ext()
   LIN {X -1.249, Y 16.640, Z 98.600}
   LaserStart_Ext()
   LIN {X 7.845, Y 16.640, Z 98.600}
   LaserEnd_Ext()
   LIN {X 7.592, Y 17.640, Z 98.600}
   LaserStart_Ext()
   LIN {X -1.343, Y 17.640, Z 98.600}
   LaserEnd_Ext()
   LIN {X -1.492, Y 18.640, Z 98.600}
   LaserStart_Ext()
   LIN {X 7.339, Y 18.640, Z 98.600}
   LaserEnd_Ext()
   LIN {X 7.086, Y 19.640, Z 98.600}
   LaserStart_Ext()
   LIN {X -1.659, Y 19.640, Z 98.600}
   LaserEnd_Ext()
   LIN {X -1.826, Y 20.640, Z 98.600}
   LaserStart_Ext()
   LIN {X 6.778, Y 20.640, Z 98.600}
   LaserEnd_Ext()
   LIN {X 6.450, Y 21.640, Z 98.600}
   LaserStart_Ext()
   LIN {X -2.015, Y 21.640, Z 98.600}
   LaserEnd_Ext()
   LIN {X -2.233, Y 22.640, Z 98.600}
   LaserStart_Ext()
   LIN {X 6.122, Y 22.640, Z 98.600}
   LaserEnd_Ext()
   LIN {X 5.794, Y 23.640, Z 98.600}
   LaserStart_Ext()
   LIN {X -2.451, Y 23.640, Z 98.600}
   LaserEnd_Ext()
   LIN {X -2.670, Y 24.640, Z 98.600}
   LaserStart_Ext()
   LIN {X 5.452, Y 24.640, Z 98.600}
   LaserEnd_Ext()
   LIN {X 5.079, Y 25.640, Z 98.600}
   LaserStart_Ext()
   LIN {X -2.888, Y 25.640, Z 98.600}
   LaserEnd_Ext()
   LIN {X -3.114, Y 26.640, Z 98.600}
   LaserStart_Ext()
   LIN {X 4.706, Y 26.640, Z 98.600}
   LaserEnd_Ext()
   LIN {X 4.334, Y 27.640, Z 98.600}
   LaserStart_Ext()
   LIN {X -3.407, Y 27.640, Z 98.600}
   LaserEnd_Ext()
   LIN {X -3.699, Y 28.640, Z 98.600}
   LaserStart_Ext()
   LIN {X 3.961, Y 28.640, Z 98.600}
   LaserEnd_Ext()
   LIN {X 3.581, Y 29.640, Z 98.600}
   LaserStart_Ext()
   LIN {X -3.991, Y 29.640, Z 98.600}
   LaserEnd_Ext()
   LIN {X -4.325, Y 30.640, Z 98.600}
   LaserStart_Ext()
   LIN {X 3.183, Y 30.640, Z 98.600}
   LaserEnd_Ext()
   LIN {X 2.756, Y 31.640, Z 98.600}
   LaserStart_Ext()
   LIN {X -4.669, Y 31.640, Z 98.600}
   LaserEnd_Ext()
   LIN {X -5.043, Y 32.640, Z 98.600}
   LaserStart_Ext()
   LIN {X 2.285, Y 32.640, Z 98.600}
   LaserEnd_Ext()
   LIN {X 1.820, Y 33.640, Z 98.600}
   LaserStart_Ext()
   LIN {X -5.416, Y 33.640, Z 98.600}
   LaserEnd_Ext()
   LIN {X -5.789, Y 34.640, Z 98.600}
   LaserStart_Ext()
   LIN {X 1.357, Y 34.640, Z 98.600}
   LaserEnd_Ext()
   LIN {X 0.898, Y 35.640, Z 98.600}
   LaserStart_Ext()
   LIN {X -6.162, Y 35.640, Z 98.600}
   LaserEnd_Ext()
   LIN {X -6.569, Y 36.640, Z 98.600}
   LaserStart_Ext()
   LIN {X 0.438, Y 36.640, Z 98.600}
   LaserEnd_Ext()
   LIN {X -0.022, Y 37.640, Z 98.600}
   LaserStart_Ext()
   LIN {X -7.015, Y 37.640, Z 98.600}
   LaserEnd_Ext()
   LIN {X -7.463, Y 38.640, Z 98.600}
   LaserStart_Ext()
   LIN {X -0.495, Y 38.640, Z 98.600}
   LaserEnd_Ext()
   LIN {X -1.016, Y 39.640, Z 98.600}
   LaserStart_Ext()
   LIN {X -7.936, Y 39.640, Z 98.600}
   LaserEnd_Ext()
   LIN {X -8.421, Y 40.640, Z 98.600}
   LaserStart_Ext()
   LIN {X -1.548, Y 40.640, Z 98.600}
   LaserEnd_Ext()
   LIN {X -2.088, Y 41.640, Z 98.600}
   LaserStart_Ext()
   LIN {X -8.855, Y 41.640, Z 98.600}
   LaserEnd_Ext()
   LIN {X -9.093, Y 42.640, Z 98.600}
   LaserStart_Ext()
   LIN {X -2.645, Y 42.640, Z 98.600}
   LaserEnd_Ext()
   LIN {X -3.211, Y 43.640, Z 98.600}
   LaserStart_Ext()
   LIN {X -8.991, Y 43.640, Z 98.600}
   LaserEnd_Ext()
   LIN {X -8.401, Y 44.640, Z 98.600}
   LaserStart_Ext()
   LIN {X -3.915, Y 44.640, Z 98.600}
   LaserEnd_Ext()
   LIN {X -5.443, Y 45.640, Z 98.600}
   LaserStart_Ext()
   LIN {X -6.777, Y 45.640, Z 98.600}
   LaserEnd_Ext()
   LIN {X 6.360, Y -22.007, Z 99.450}
   LaserStart_Ext()
   LIN {X 5.398, Y -22.437, Z 99.450} C_DIS
   LIN {X 4.418, Y -22.881, Z 99.450} C_DIS
   LIN {X 3.725, Y -22.882, Z 99.450} C_DIS
   LIN {X 2.293, Y -22.882, Z 99.450} C_DIS
   LIN {X 0.477, Y -22.054, Z 99.450} C_DIS
   LIN {X 0.377, Y -21.985, Z 99.450} C_DIS
   LIN {X -0.970, Y -20.466, Z 99.450} C_DIS
   LIN {X -1.548, Y -18.589, Z 99.450} C_DIS
   LIN {X -1.584, Y -18.472, Z 99.450} C_DIS
   LIN {X -1.545, Y -18.303, Z 99.450} C_DIS
   LIN {X -0.902, Y -15.461, Z 99.450} C_DIS
   LIN {X 0.363, Y -14.065, Z 99.450} C_DIS
   LIN {X 0.475, Y -13.940, Z 99.450} C_DIS
   LIN {X 0.710, Y -13.834, Z 99.450} C_DIS
   LIN {X 2.349, Y -13.099, Z 99.450} C_DIS
   LIN {X 3.714, Y -13.093, Z 99.450} C_DIS
   LIN {X 4.500, Y -13.088, Z 99.450} C_DIS
   LIN {X 5.426, Y -13.513, Z 99.450} C_DIS
   LIN {X 6.430, Y -13.977, Z 99.450} C_DIS
   LIN {X 7.140, Y -14.882, Z 99.450} C_DIS
   LIN {X 8.003, Y -15.975, Z 99.450} C_DIS
   LIN {X 8.217, Y -17.119, Z 99.450} C_DIS
   LIN {X 8.405, Y -18.148, Z 99.450} C_DIS
   LIN {X 8.157, Y -19.006, Z 99.450} C_DIS
   LIN {X 7.769, Y -20.398, Z 99.450} C_DIS
   LIN {X 6.820, Y -21.492, Z 99.450} C_DIS
   LIN {X 6.360, Y -22.007, Z 99.450}
   LaserEnd_Ext()
   LIN {X -1.931, Y 0.089, Z 99.450}
   LaserStart_Ext()
   LIN {X -1.873, Y 0.710, Z 99.450} C_DIS
   LIN {X -1.595, Y 8.225, Z 99.450} C_DIS
   LIN {X -1.600, Y 9.659, Z 99.450} C_DIS
   LIN {X -2.408, Y 18.243, Z 99.450} C_DIS
   LIN {X -2.713, Y 20.072, Z 99.450} C_DIS
   LIN {X -4.093, Y 26.397, Z 99.450} C_DIS
   LIN {X -4.883, Y 29.102, Z 99.450} C_DIS
   LIN {X -5.808, Y 31.790, Z 99.450} C_DIS
   LIN {X -7.133, Y 35.339, Z 99.450} C_DIS
   LIN {X -7.375, Y 35.908, Z 99.450} C_DIS
   LIN {X -7.542, Y 36.304, Z 99.450} C_DIS
   LIN {X -8.180, Y 37.724, Z 99.450} C_DIS
   LIN {X -8.498, Y 38.428, Z 99.450} C_DIS
   LIN {X -8.830, Y 39.114, Z 99.450} C_DIS
   LIN {X -9.193, Y 39.869, Z 99.450} C_DIS
   LIN {X -9.440, Y 40.370, Z 99.450} C_DIS
   LIN {X -9.747, Y 40.990, Z 99.450} C_DIS
   LIN {X -10.033, Y 41.822, Z 99.450} C_DIS
   LIN {X -10.158, Y 42.204, Z 99.450} C_DIS
   LIN {X -10.128, Y 42.690, Z 99.450} C_DIS
   LIN {X -10.065, Y 43.891, Z 99.450} C_DIS
   LIN {X -9.466, Y 45.063, Z 99.450} C_DIS
   LIN {X -9.342, Y 45.306, Z 99.450} C_DIS
   LIN {X -9.189, Y 45.399, Z 99.450} C_DIS
   LIN {X -7.060, Y 46.718, Z 99.450} C_DIS
   LIN {X -5.919, Y 46.703, Z 99.450} C_DIS
   LIN {X -5.315, Y 46.696, Z 99.450} C_DIS
   LIN {X -5.001, Y 46.545, Z 99.450} C_DIS
   LIN {X -3.749, Y 45.937, Z 99.450} C_DIS
   LIN {X -2.782, Y 44.835, Z 99.450} C_DIS
   LIN {X -2.035, Y 43.539, Z 99.450} C_DIS
   LIN {X -1.369, Y 42.351, Z 99.450} C_DIS
   LIN {X -1.099, Y 41.868, Z 99.450} C_DIS
   LIN {X -0.004, Y 39.807, Z 99.450} C_DIS
   LIN {X 0.231, Y 39.366, Z 99.450} C_DIS
   LIN {X 0.488, Y 38.872, Z 99.450} C_DIS
   LIN {X 1.331, Y 37.038, Z 99.450} C_DIS
   LIN {X 2.948, Y 33.559, Z 99.450} C_DIS
   LIN {X 3.771, Y 31.832, Z 99.450} C_DIS
   LIN {X 5.169, Y 28.314, Z 99.450} C_DIS
   LIN {X 6.403, Y 25.003, Z 99.450} C_DIS
   LIN {X 8.059, Y 19.955, Z 99.450} C_DIS
   LIN {X 8.863, Y 16.782, Z 99.450} C_DIS
   LIN {X 10.349, Y 10.853, Z 99.450} C_DIS
   LIN {X 11.126, Y 6.103, Z 99.450} C_DIS
   LIN {X 11.821, Y 1.845, Z 99.450} C_DIS
   LIN {X 12.268, Y -2.687, Z 99.450} C_DIS
   LIN {X 12.316, Y -3.281, Z 99.450} C_DIS
   LIN {X 12.407, Y -5.183, Z 99.450} C_DIS
   LIN {X 12.581, Y -8.471, Z 99.450} C_DIS
   LIN {X 12.605, Y -10.151, Z 99.450} C_DIS
   LIN {X 12.620, Y -12.275, Z 99.450} C_DIS
   LIN {X 12.561, Y -15.172, Z 99.450} C_DIS
   LIN {X 12.553, Y -15.350, Z 99.450} C_DIS
   LIN {X 12.399, Y -18.492, Z 99.450} C_DIS
   LIN {X 12.025, Y -20.129, Z 99.450} C_DIS
   LIN {X 11.731, Y -21.377, Z 99.450} C_DIS
   LIN {X 10.160, Y -23.640, Z 99.450} C_DIS
   LIN {X 9.523, Y -24.563, Z 99.450} C_DIS
   LIN {X 9.095, Y -24.849, Z 99.450} C_DIS
   LIN {X 6.692, Y -26.354, Z 99.450} C_DIS
   LIN {X 4.373, Y -26.781, Z 99.450} C_DIS
   LIN {X 2.802, Y -26.919, Z 99.450} C_DIS
   LIN {X 0.206, Y -26.444, Z 99.450} C_DIS
   LIN {X -0.197, Y -26.190, Z 99.450} C_DIS
   LIN {X -3.016, Y -24.371, Z 99.450} C_DIS
   LIN {X -4.555, Y -22.199, Z 99.450} C_DIS
   LIN {X -4.715, Y -21.977, Z 99.450} C_DIS
   LIN {X -4.827, Y -21.531, Z 99.450} C_DIS
   LIN {X -5.610, Y -18.376, Z 99.450} C_DIS
   LIN {X -5.231, Y -15.682, Z 99.450} C_DIS
   LIN {X -5.170, Y -15.236, Z 99.450} C_DIS
   LIN {X -5.033, Y -14.785, Z 99.450} C_DIS
   LIN {X -4.295, Y -12.375, Z 99.450} C_DIS
   LIN {X -3.810, Y -10.429, Z 99.450} C_DIS
   LIN {X -3.096, Y -7.481, Z 99.450} C_DIS
   LIN {X -2.679, Y -5.072, Z 99.450} C_DIS
   LIN {X -2.016, Y -0.621, Z 99.450} C_DIS
   LIN {X -1.951, Y -0.069, Z 99.450} C_DIS
   LIN {X -1.931, Y 0.089, Z 99.450}
   LaserEnd_Ext()
   LIN {X 11.602, Y -13.140, Z 99.450}
   LaserStart_Ext()
   LIN {X 11.602, Y -9.956, Z 99.450}
   LaserEnd_Ext()
   LIN {X 10.602, Y 3.104, Z 99.450}
   LaserStart_Ext()
   LIN {X 10.602, Y -21.249, Z 99.450}
   LaserEnd_Ext()
   LIN {X 9.602, Y -22.690, Z 99.450}
   LaserStart_Ext()
   LIN {X 9.602, Y 9.223, Z 99.450}
   LaserEnd_Ext()
   LIN {X 8.602, Y 13.709, Z 99.450}
   LaserStart_Ext()
   LIN {X 8.602, Y -15.120, Z 99.450}
   LaserEnd_Ext()
   LIN {X 8.602, Y -20.950, Z 99.450}
   LaserStart_Ext()
   LIN {X 8.602, Y -23.976, Z 99.450}
   LaserEnd_Ext()
   LIN {X 7.602, Y -24.604, Z 99.450}
   LaserStart_Ext()
   LIN {X 7.602, Y -22.117, Z 99.450}
   LaserEnd_Ext()
   LIN {X 7.602, Y -13.851, Z 99.450}
   LaserStart_Ext()
   LIN {X 7.602, Y 17.687, Z 99.450}
   LaserEnd_Ext()
   LIN {X 6.602, Y 21.189, Z 99.450}
   LaserStart_Ext()
   LIN {X 6.602, Y -12.955, Z 99.450}
   LaserEnd_Ext()
   LIN {X 6.602, Y -22.994, Z 99.450}
   LaserStart_Ext()
   LIN {X 6.602, Y -25.230, Z 99.450}
   LaserEnd_Ext()
   LIN {X 5.602, Y -25.538, Z 99.450}
   LaserStart_Ext()
   LIN {X 5.602, Y -23.442, Z 99.450}
   LaserEnd_Ext()
   LIN {X 5.602, Y -12.493, Z 99.450}
   LaserStart_Ext()
   LIN {X 5.602, Y 24.236, Z 99.450}
   LaserEnd_Ext()
   LIN {X 4.602, Y 26.972, Z 99.450}
   LaserStart_Ext()
   LIN {X 4.602, Y -12.093, Z 99.450}
   LaserEnd_Ext()
   LIN {X 4.602, Y -23.862, Z 99.450}
   LaserStart_Ext()
   LIN {X 4.602, Y -25.722, Z 99.450}
   LaserEnd_Ext()
   LIN {X 3.602, Y -25.845, Z 99.450}
   LaserStart_Ext()
   LIN {X 3.602, Y -23.882, Z 99.450}
   LaserEnd_Ext()
   LIN {X 3.602, Y -12.093, Z 99.450}
   LaserStart_Ext()
   LIN {X 3.602, Y 29.550, Z 99.450}
   LaserEnd_Ext()
   LIN {X 2.602, Y 31.962, Z 99.450}
   LaserStart_Ext()
   LIN {X 2.602, Y -12.098, Z 99.450}
   LaserEnd_Ext()
   LIN {X 2.602, Y -23.882, Z 99.450}
   LaserStart_Ext()
   LIN {X 2.602, Y -25.866, Z 99.450}
   LaserEnd_Ext()
   LIN {X 1.602, Y -25.683, Z 99.450}
   LaserStart_Ext()
   LIN {X 1.602, Y -23.666, Z 99.450}
   LaserEnd_Ext()
   LIN {X 1.602, Y -12.338, Z 99.450}
   LaserStart_Ext()
   LIN {X 1.602, Y 34.083, Z 99.450}
   LaserEnd_Ext()
   LIN {X 0.602, Y 36.234, Z 99.450}
   LaserStart_Ext()
   LIN {X 0.602, Y -12.787, Z 99.450}
   LaserEnd_Ext()
   LIN {X 0.602, Y -23.210, Z 99.450}
   LaserStart_Ext()
   LIN {X 0.602, Y -25.500, Z 99.450}
   LaserEnd_Ext()
   LIN {X -0.398, Y -24.870, Z 99.450}
   LaserStart_Ext()
   LIN {X -0.398, Y -22.618, Z 99.450}
   LaserEnd_Ext()
   LIN {X -0.398, Y -13.415, Z 99.450}
   LaserStart_Ext()
   LIN {X -0.398, Y 38.405, Z 99.450}
   LaserEnd_Ext()
   LIN {X -1.398, Y 40.300, Z 99.450}
   LaserStart_Ext()
   LIN {X -1.398, Y 18.187, Z 99.450}
   LaserEnd_Ext()
   LIN {X -1.398, Y -3.261, Z 99.450}
   LaserStart_Ext()
   LIN {X -1.398, Y -14.519, Z 99.450}
   LaserEnd_Ext()
   LIN {X -1.398, Y -21.491, Z 99.450}
   LaserStart_Ext()
   LIN {X -1.398, Y -24.225, Z 99.450}
   LaserEnd_Ext()
   LIN {X -2.398, Y -23.513, Z 99.450}
   LaserStart_Ext()
   LIN {X -2.398, Y -19.227, Z 99.450}
   LaserEnd_Ext()
   LIN {X -2.398, Y -17.541, Z 99.450}
   LaserStart_Ext()
   LIN {X -2.398, Y -8.847, Z 99.450}
   LaserEnd_Ext()
   LIN {X -2.398, Y 23.320, Z 99.450}
   LaserStart_Ext()
   LIN {X -2.398, Y 42.142, Z 99.450}
   LaserEnd_Ext()
   LIN {X -3.398, Y 43.903, Z 99.450}
   LaserStart_Ext()
   LIN {X -3.398, Y 27.584, Z 99.450}
   LaserEnd_Ext()
   LIN {X -3.398, Y -12.861, Z 99.450}
   LaserStart_Ext()
   LIN {X -3.398, Y -22.102, Z 99.450}
   LaserEnd_Ext()
   LIN {X -4.398, Y -19.108, Z 99.450}
   LaserStart_Ext()
   LIN {X -4.398, Y -16.941, Z 99.450}
   LaserEnd_Ext()
   LIN {X -4.398, Y 30.764, Z 99.450}
   LaserStart_Ext()
   LIN {X -4.398, Y 45.140, Z 99.450}
   LaserEnd_Ext()
   LIN {X -5.398, Y 45.626, Z 99.450}
   LaserStart_Ext()
   LIN {X -5.398, Y 33.550, Z 99.450}
   LaserEnd_Ext()
   LIN {X -6.398, Y 36.166, Z 99.450}
   LaserStart_Ext()
   LIN {X -6.398, Y 45.709, Z 99.450}
   LaserEnd_Ext()
   LIN {X -7.398, Y 45.332, Z 99.450}
   LaserStart_Ext()
   LIN {X -7.398, Y 38.422, Z 99.450}
   LaserEnd_Ext()
   LIN {X -8.398, Y 40.518, Z 99.450}
   LaserStart_Ext()
   LIN {X -8.398, Y 44.713, Z 99.450}
   LaserEnd_Ext()
   LIN {X 8.080, Y -15.905, Z 100.300}
   LaserStart_Ext()
   LIN {X 8.395, Y -17.595, Z 100.300} C_DIS
   LIN {X 8.486, Y -18.077, Z 100.300} C_DIS
   LIN {X 8.284, Y -18.819, Z 100.300} C_DIS
   LIN {X 7.871, Y -20.303, Z 100.300} C_DIS
   LIN {X 7.072, Y -21.224, Z 100.300} C_DIS
   LIN {X 6.468, Y -21.929, Z 100.300} C_DIS
   LIN {X 5.956, Y -22.164, Z 100.300} C_DIS
   LIN {X 4.504, Y -22.821, Z 100.300} C_DIS
   LIN {X 2.555, Y -22.826, Z 100.300} C_DIS
   LIN {X 2.387, Y -22.826, Z 100.300} C_DIS
   LIN {X 2.174, Y -22.729, Z 100.300} C_DIS
   LIN {X 0.504, Y -21.973, Z 100.300} C_DIS
   LIN {X -0.419, Y -20.941, Z 100.300} C_DIS
   LIN {X -0.883, Y -20.418, Z 100.300} C_DIS
   LIN {X -1.106, Y -19.693, Z 100.300} C_DIS
   LIN {X -1.501, Y -18.425, Z 100.300} C_DIS
   LIN {X -1.085, Y -16.581, Z 100.300} C_DIS
   LIN {X -0.817, Y -15.396, Z 100.300} C_DIS
   LIN {X -0.345, Y -14.875, Z 100.300} C_DIS
   LIN {X 0.539, Y -13.894, Z 100.300} C_DIS
   LIN {X 2.387, Y -13.059, Z 100.300} C_DIS
   LIN {X 4.569, Y -13.026, Z 100.300} C_DIS
   LIN {X 6.071, Y -13.715, Z 100.300} C_DIS
   LIN {X 6.502, Y -13.911, Z 100.300} C_DIS
   LIN {X 6.902, Y -14.414, Z 100.300} C_DIS
   LIN {X 8.080, Y -15.905, Z 100.300}
   LaserEnd_Ext()
   LIN {X -2.522, Y 19.123, Z 100.300}
   LaserStart_Ext()
   LIN {X -4.135, Y 26.515, Z 100.300} C_DIS
   LIN {X -4.764, Y 28.665, Z 100.300} C_DIS
   LIN {X -6.012, Y 32.291, Z 100.300} C_DIS
   LIN {X -7.045, Y 35.062, Z 100.300} C_DIS
   LIN {X -7.234, Y 35.506, Z 100.300} C_DIS
   LIN {X -7.521, Y 36.185, Z 100.300} C_DIS
   LIN {X -7.586, Y 36.338, Z 100.300} C_DIS
   LIN {X -7.875, Y 36.974, Z 100.300} C_DIS
   LIN {X -8.546, Y 38.460, Z 100.300} C_DIS
   LIN {X -8.889, Y 39.169, Z 100.300} C_DIS
   LIN {X -9.245, Y 39.899, Z 100.300} C_DIS
   LIN {X -9.685, Y 40.784, Z 100.300} C_DIS
   LIN {X -9.801, Y 41.019, Z 100.300} C_DIS
   LIN {X -9.869, Y 41.216, Z 100.300} C_DIS
   LIN {X -10.218, Y 42.248, Z 100.300} C_DIS
   LIN {X -10.142, Y 43.582, Z 100.300} C_DIS
   LIN {X -10.125, Y 43.921, Z 100.300} C_DIS
   LIN {X -9.996, Y 44.172, Z 100.300} C_DIS
   LIN {X -9.378, Y 45.369, Z 100.300} C_DIS
   LIN {X -7.909, Y 46.276, Z 100.300} C_DIS
   LIN {X -7.127, Y 46.752, Z 100.300} C_DIS
   LIN {X -6.361, Y 46.746, Z 100.300} C_DIS
   LIN {X -5.382, Y 46.735, Z 100.300} C_DIS
   LIN {X -3.923, Y 46.032, Z 100.300} C_DIS
   LIN {X -3.815, Y 45.980, Z 100.300} C_DIS
   LIN {X -2.842, Y 44.875, Z 100.300} C_DIS
   LIN {X -2.198, Y 43.765, Z 100.300} C_DIS
   LIN {X -2.091, Y 43.579, Z 100.300} C_DIS
   LIN {X -1.903, Y 43.244, Z 100.300} C_DIS
   LIN {X -1.088, Y 41.795, Z 100.300} C_DIS
   LIN {X 0.247, Y 39.281, Z 100.300} C_DIS
   LIN {X 0.482, Y 38.838, Z 100.300} C_DIS
   LIN {X 2.509, Y 34.477, Z 100.300} C_DIS
   LIN {X 3.691, Y 31.999, Z 100.300} C_DIS
   LIN {X 5.697, Y 26.948, Z 100.300} C_DIS
   LIN {X 6.295, Y 25.345, Z 100.300} C_DIS
   LIN {X 8.142, Y 19.717, Z 100.300} C_DIS
   LIN {X 8.606, Y 17.881, Z 100.300} C_DIS
   LIN {X 10.428, Y 10.614, Z 100.300} C_DIS
   LIN {X 11.380, Y 4.791, Z 100.300} C_DIS
   LIN {X 11.871, Y 1.785, Z 100.300} C_DIS
   LIN {X 12.318, Y -2.747, Z 100.300} C_DIS
   LIN {X 12.363, Y -3.196, Z 100.300} C_DIS
   LIN {X 12.390, Y -3.692, Z 100.300} C_DIS
   LIN {X 12.639, Y -8.391, Z 100.300} C_DIS
   LIN {X 12.681, Y -11.361, Z 100.300} C_DIS
   LIN {X 12.687, Y -12.195, Z 100.300} C_DIS
   LIN {X 12.663, Y -13.394, Z 100.300} C_DIS
   LIN {X 12.633, Y -15.155, Z 100.300} C_DIS
   LIN {X 12.584, Y -16.308, Z 100.300} C_DIS
   LIN {X 12.481, Y -18.413, Z 100.300} C_DIS
   LIN {X 11.830, Y -21.253, Z 100.300} C_DIS
   LIN {X 11.762, Y -21.383, Z 100.300} C_DIS
   LIN {X 9.618, Y -24.490, Z 100.300} C_DIS
   LIN {X 8.176, Y -25.453, Z 100.300} C_DIS
   LIN {X 6.939, Y -26.228, Z 100.300} C_DIS
   LIN {X 5.746, Y -26.447, Z 100.300} C_DIS
   LIN {X 2.251, Y -26.755, Z 100.300} C_DIS
   LIN {X 0.341, Y -26.405, Z 100.300} C_DIS
   LIN {X -1.365, Y -25.331, Z 100.300} C_DIS
   LIN {X -2.920, Y -24.327, Z 100.300} C_DIS
   LIN {X -3.770, Y -23.128, Z 100.300} C_DIS
   LIN {X -4.626, Y -21.936, Z 100.300} C_DIS
   LIN {X -5.228, Y -19.551, Z 100.300} C_DIS
   LIN {X -5.529, Y -18.338, Z 100.300} C_DIS
   LIN {X -5.383, Y -17.303, Z 100.300} C_DIS
   LIN {X -5.096, Y -15.197, Z 100.300} C_DIS
   LIN {X -4.453, Y -13.072, Z 100.300} C_DIS
   LIN {X -4.234, Y -12.357, Z 100.300} C_DIS
   LIN {X -4.090, Y -11.781, Z 100.300} C_DIS
   LIN {X -3.046, Y -7.462, Z 100.300} C_DIS
   LIN {X -2.852, Y -6.343, Z 100.300} C_DIS
   LIN {X -1.917, Y -0.074, Z 100.300} C_DIS
   LIN {X -1.896, Y 0.103, Z 100.300} C_DIS
   LIN {X -1.872, Y 0.352, Z 100.300} C_DIS
   LIN {X -1.567, Y 8.576, Z 100.300} C_DIS
   LIN {X -1.570, Y 9.299, Z 100.300} C_DIS
   LIN {X -2.458, Y 18.739, Z 100.300} C_DIS
   LIN {X -2.522, Y 19.123, Z 100.300}
   LaserEnd_Ext()
   LIN {X -7.225, Y 45.522, Z 100.300}
   LaserStart_Ext()
   LIN {X -5.168, Y 45.522, Z 100.300}
   LaserEnd_Ext()
   LIN {X -3.863, Y 44.522, Z 100.300}
   LaserStart_Ext()
   LIN {X -8.690, Y 44.522, Z 100.300}
   LaserEnd_Ext()
   LIN {X -9.144, Y 43.522, Z 100.300}
   LaserStart_Ext()
   LIN {X -3.213, Y 43.522, Z 100.300}
   LaserEnd_Ext()
   LIN {X -2.644, Y 42.522, Z 100.300}
   LaserStart_Ext()
   LIN {X -9.201, Y 42.522, Z 100.300}
   LaserEnd_Ext()
   LIN {X -8.917, Y 41.522, Z 100.300}
   LaserStart_Ext()
   LIN {X -2.081, Y 41.522, Z 100.300}
   LaserEnd_Ext()
   LIN {X -1.544, Y 40.522, Z 100.300}
   LaserStart_Ext()
   LIN {X -8.438, Y 40.522, Z 100.300}
   LaserEnd_Ext()
   LIN {X -7.949, Y 39.522, Z 100.300}
   LaserStart_Ext()
   LIN {X -1.013, Y 39.522, Z 100.300}
   LaserEnd_Ext()
   LIN {X -0.482, Y 38.522, Z 100.300}
   LaserStart_Ext()
   LIN {X -7.477, Y 38.522, Z 100.300}
   LaserEnd_Ext()
   LIN {X -7.025, Y 37.522, Z 100.300}
   LaserStart_Ext()
   LIN {X -0.009, Y 37.522, Z 100.300}
   LaserEnd_Ext()
   LIN {X 0.456, Y 36.522, Z 100.300}
   LaserStart_Ext()
   LIN {X -6.578, Y 36.522, Z 100.300}
   LaserEnd_Ext()
   LIN {X -6.154, Y 35.522, Z 100.300}
   LaserStart_Ext()
   LIN {X 0.921, Y 35.522, Z 100.300}
   LaserEnd_Ext()
   LIN {X 1.386, Y 34.522, Z 100.300}
   LaserStart_Ext()
   LIN {X -5.777, Y 34.522, Z 100.300}
   LaserEnd_Ext()
   LIN {X -5.403, Y 33.522, Z 100.300}
   LaserStart_Ext()
   LIN {X 1.857, Y 33.522, Z 100.300}
   LaserEnd_Ext()
   LIN {X 2.334, Y 32.522, Z 100.300}
   LaserStart_Ext()
   LIN {X -5.033, Y 32.522, Z 100.300}
   LaserEnd_Ext()
   LIN {X -4.689, Y 31.522, Z 100.300}
   LaserStart_Ext()
   LIN {X 2.804, Y 31.522, Z 100.300}
   LaserEnd_Ext()
   LIN {X 3.202, Y 30.522, Z 100.300}
   LaserStart_Ext()
   LIN {X -4.345, Y 30.522, Z 100.300}
   LaserEnd_Ext()
   LIN {X -4.001, Y 29.522, Z 100.300}
   LaserStart_Ext()
   LIN {X 3.599, Y 29.522, Z 100.300}
   LaserEnd_Ext()
   LIN {X 3.996, Y 28.522, Z 100.300}
   LaserStart_Ext()
   LIN {X -3.680, Y 28.522, Z 100.300}
   LaserEnd_Ext()
   LIN {X -3.388, Y 27.522, Z 100.300}
   LaserStart_Ext()
   LIN {X 4.393, Y 27.522, Z 100.300}
   LaserEnd_Ext()
   LIN {X 4.789, Y 26.522, Z 100.300}
   LaserStart_Ext()
   LIN {X -3.113, Y 26.522, Z 100.300}
   LaserEnd_Ext()
   LIN {X -2.895, Y 25.522, Z 100.300}
   LaserStart_Ext()
   LIN {X 5.161, Y 25.522, Z 100.300}
   LaserEnd_Ext()
   LIN {X 5.512, Y 24.522, Z 100.300}
   LaserStart_Ext()
   LIN {X -2.677, Y 24.522, Z 100.300}
   LaserEnd_Ext()
   LIN {X -2.459, Y 23.522, Z 100.300}
   LaserStart_Ext()
   LIN {X 5.840, Y 23.522, Z 100.300}
   LaserEnd_Ext()
   LIN {X 6.169, Y 22.522, Z 100.300}
   LaserStart_Ext()
   LIN {X -2.240, Y 22.522, Z 100.300}
   LaserEnd_Ext()
   LIN {X -2.022, Y 21.522, Z 100.300}
   LaserStart_Ext()
   LIN {X 6.497, Y 21.522, Z 100.300}
   LaserEnd_Ext()
   LIN {X 6.825, Y 20.522, Z 100.300}
   LaserStart_Ext()
   LIN {X -1.804, Y 20.522, Z 100.300}
   LaserEnd_Ext()
   LIN {X -1.586, Y 19.522, Z 100.300}
   LaserStart_Ext()
   LIN {X 7.153, Y 19.522, Z 100.300}
   LaserEnd_Ext()
   LIN {X 7.413, Y 18.522, Z 100.300}
   LaserStart_Ext()
   LIN {X -1.433, Y 18.522, Z 100.300}
   LaserEnd_Ext()
   LIN {X -1.339, Y 17.522, Z 100.300}
   LaserStart_Ext()
   LIN {X 7.665, Y 17.522, Z 100.300}
   LaserEnd_Ext()
   LIN {X 7.916, Y 16.522, Z 100.300}
   LaserStart_Ext()
   LIN {X -1.245, Y 16.522, Z 100.300}
   LaserEnd_Ext()
   LIN {X -1.151, Y 15.522, Z 100.300}
   LaserStart_Ext()
   LIN {X 8.167, Y 15.522, Z 100.300}
   LaserEnd_Ext()
   LIN {X 8.417, Y 14.522, Z 100.300}
   LaserStart_Ext()
   LIN {X -1.057, Y 14.522, Z 100.300}
   LaserEnd_Ext()
   LIN {X -0.963, Y 13.522, Z 100.300}
   LaserStart_Ext()
   LIN {X 8.668, Y 13.522, Z 100.300}
   LaserEnd_Ext()
   LIN {X 8.919, Y 12.522, Z 100.300}
   LaserStart_Ext()
   LIN {X -0.869, Y 12.522, Z 100.300}
   LaserEnd_Ext()
   LIN {X -0.775, Y 11.522, Z 100.300}
   LaserStart_Ext()
   LIN {X 9.169, Y 11.522, Z 100.300}
   LaserEnd_Ext()
   LIN {X 9.420, Y 10.522, Z 100.300}
   LaserStart_Ext()
   LIN {X -0.681, Y 10.522, Z 100.300}
   LaserEnd_Ext()
   LIN {X -0.587, Y 9.522, Z 100.300}
   LaserStart_Ext()
   LIN {X 9.593, Y 9.522, Z 100.300}
   LaserEnd_Ext()
   LIN {X 9.757, Y 8.522, Z 100.300}
   LaserStart_Ext()
   LIN {X -0.569, Y 8.522, Z 100.300}
   LaserEnd_Ext()
   LIN {X -0.606, Y 7.522, Z 100.300}
   LaserStart_Ext()
   LIN {X 9.920, Y 7.522, Z 100.300}
   LaserEnd_Ext()
   LIN {X 10.084, Y 6.522, Z 100.300}
   LaserStart_Ext()
   LIN {X -0.643, Y 6.522, Z 100.300}
   LaserEnd_Ext()
   LIN {X -0.680, Y 5.522, Z 100.300}
   LaserStart_Ext()
   LIN {X 10.247, Y 5.522, Z 100.300}
   LaserEnd_Ext()
   LIN {X 10.411, Y 4.522, Z 100.300}
   LaserStart_Ext()
   LIN {X -0.717, Y 4.522, Z 100.300}
   LaserEnd_Ext()
   LIN {X -0.754, Y 3.522, Z 100.300}
   LaserStart_Ext()
   LIN {X 10.574, Y 3.522, Z 100.300}
   LaserEnd_Ext()
   LIN {X 10.737, Y 2.522, Z 100.300}
   LaserStart_Ext()
   LIN {X -0.791, Y 2.522, Z 100.300}
   LaserEnd_Ext()
   LIN {X -0.828, Y 1.522, Z 100.300}
   LaserStart_Ext()
   LIN {X 10.892, Y 1.522, Z 100.300}
   LaserEnd_Ext()
   LIN {X 10.991, Y 0.522, Z 100.300}
   LaserStart_Ext()
   LIN {X -0.865, Y 0.522, Z 100.300}
   LaserEnd_Ext()
   LIN {X -0.967, Y -0.478, Z 100.300}
   LaserStart_Ext()
   LIN {X 11.089, Y -0.478, Z 100.300}
   LaserEnd_Ext()
   LIN {X 11.188, Y -1.478, Z 100.300}
   LaserStart_Ext()
   LIN {X -1.116, Y -1.478, Z 100.300}
   LaserEnd_Ext()
   LIN {X -1.265, Y -2.478, Z 100.300}
   LaserStart_Ext()
   LIN {X 11.287, Y -2.478, Z 100.300}
   LaserEnd_Ext()
   LIN {X 11.377, Y -3.478, Z 100.300}
   LaserStart_Ext()
   LIN {X -1.414, Y -3.478, Z 100.300}
   LaserEnd_Ext()
   LIN {X -1.563, Y -4.478, Z 100.300}
   LaserStart_Ext()
   LIN {X 11.430, Y -4.478, Z 100.300}
   LaserEnd_Ext()
   LIN {X 11.483, Y -5.478, Z 100.300}
   LaserStart_Ext()
   LIN {X -1.712, Y -5.478, Z 100.300}
   LaserEnd_Ext()
   LIN {X -1.861, Y -6.478, Z 100.300}
   LaserStart_Ext()
   LIN {X 11.537, Y -6.478, Z 100.300}
   LaserEnd_Ext()
   LIN {X 11.590, Y -7.478, Z 100.300}
   LaserStart_Ext()
   LIN {X -2.034, Y -7.478, Z 100.300}
   LaserEnd_Ext()
   LIN {X -2.263, Y -8.478, Z 100.300}
   LaserStart_Ext()
   LIN {X 11.640, Y -8.478, Z 100.300}
   LaserEnd_Ext()
   LIN {X 11.655, Y -9.478, Z 100.300}
   LaserStart_Ext()
   LIN {X -2.505, Y -9.478, Z 100.300}
   LaserEnd_Ext()
   LIN {X -2.746, Y -10.478, Z 100.300}
   LaserStart_Ext()
   LIN {X 11.669, Y -10.478, Z 100.300}
   LaserEnd_Ext()
   LIN {X 11.682, Y -11.478, Z 100.300}
   LaserStart_Ext()
   LIN {X -2.988, Y -11.478, Z 100.300}
   LaserEnd_Ext()
   LIN {X -3.234, Y -12.478, Z 100.300}
   LaserStart_Ext()
   LIN {X 1.243, Y -12.478, Z 100.300}
   LaserEnd_Ext()
   LIN {X 5.773, Y -12.478, Z 100.300}
   LaserStart_Ext()
   LIN {X 11.681, Y -12.478, Z 100.300}
   LaserEnd_Ext()
   LIN {X 11.661, Y -13.478, Z 100.300}
   LaserStart_Ext()
   LIN {X 7.435, Y -13.478, Z 100.300}
   LaserEnd_Ext()
   LIN {X -0.432, Y -13.478, Z 100.300}
   LaserStart_Ext()
   LIN {X -3.531, Y -13.478, Z 100.300}
   LaserEnd_Ext()
   LIN {X -3.834, Y -14.478, Z 100.300}
   LaserStart_Ext()
   LIN {X -1.335, Y -14.478, Z 100.300}
   LaserEnd_Ext()
   LIN {X 8.227, Y -14.478, Z 100.300}
   LaserStart_Ext()
   LIN {X 11.644, Y -14.478, Z 100.300}
   LaserEnd_Ext()
   LIN {X 11.618, Y -15.478, Z 100.300}
   LaserStart_Ext()
   LIN {X 8.983, Y -15.478, Z 100.300}
   LaserEnd_Ext()
   LIN {X -1.861, Y -15.478, Z 100.300}
   LaserStart_Ext()
   LIN {X -4.125, Y -15.478, Z 100.300}
   LaserEnd_Ext()
   LIN {X -4.261, Y -16.478, Z 100.300}
   LaserStart_Ext()
   LIN {X -2.087, Y -16.478, Z 100.300}
   LaserEnd_Ext()
   LIN {X 9.204, Y -16.478, Z 100.300}
   LaserStart_Ext()
   LIN {X 11.574, Y -16.478, Z 100.300}
   LaserEnd_Ext()
   LIN {X 11.525, Y -17.478, Z 100.300}
   LaserStart_Ext()
   LIN {X 9.391, Y -17.478, Z 100.300}
   LaserEnd_Ext()
   LIN {X -2.313, Y -17.478, Z 100.300}
   LaserStart_Ext()
   LIN {X -4.398, Y -17.478, Z 100.300}
   LaserEnd_Ext()
   LIN {X -4.464, Y -18.478, Z 100.300}
   LaserStart_Ext()
   LIN {X -2.499, Y -18.478, Z 100.300}
   LaserEnd_Ext()
   LIN {X 9.414, Y -18.478, Z 100.300}
   LaserStart_Ext()
   LIN {X 11.440, Y -18.478, Z 100.300}
   LaserEnd_Ext()
   LIN {X 11.211, Y -19.478, Z 100.300}
   LaserStart_Ext()
   LIN {X 9.138, Y -19.478, Z 100.300}
   LaserEnd_Ext()
   LIN {X -2.220, Y -19.478, Z 100.300}
   LaserStart_Ext()
   LIN {X -4.215, Y -19.478, Z 100.300}
   LaserEnd_Ext()
   LIN {X -3.962, Y -20.478, Z 100.300}
   LaserStart_Ext()
   LIN {X -1.910, Y -20.478, Z 100.300}
   LaserEnd_Ext()
   LIN {X 8.860, Y -20.478, Z 100.300}
   LaserStart_Ext()
   LIN {X 10.982, Y -20.478, Z 100.300}
   LaserEnd_Ext()
   LIN {X 10.481, Y -21.478, Z 100.300}
   LaserStart_Ext()
   LIN {X 8.175, Y -21.478, Z 100.300}
   LaserEnd_Ext()
   LIN {X -1.279, Y -21.478, Z 100.300}
   LaserStart_Ext()
   LIN {X -3.710, Y -21.478, Z 100.300}
   LaserEnd_Ext()
   LIN {X -3.006, Y -22.478, Z 100.300}
   LaserStart_Ext()
   LIN {X -0.386, Y -22.478, Z 100.300}
   LaserEnd_Ext()
   LIN {X 7.314, Y -22.478, Z 100.300}
   LaserStart_Ext()
   LIN {X 9.791, Y -22.478, Z 100.300}
   LaserEnd_Ext()
   LIN {X 9.101, Y -23.478, Z 100.300}
   LaserStart_Ext()
   LIN {X 5.477, Y -23.478, Z 100.300}
   LaserEnd_Ext()
   LIN {X 1.405, Y -23.478, Z 100.300}
   LaserStart_Ext()
   LIN {X -2.296, Y -23.478, Z 100.300}
   LaserEnd_Ext()
   LIN {X -0.842, Y -24.478, Z 100.300}
   LaserStart_Ext()
   LIN {X 7.835, Y -24.478, Z 100.300}
   LaserEnd_Ext()
   LIN {X 5.350, Y -25.478, Z 100.300}
   LaserStart_Ext()
   LIN {X 0.832, Y -25.478, Z 100.300}
   LaserEnd_Ext()
   LIN {X 8.156, Y -15.835, Z 101.150}
   LaserStart_Ext()
   LIN {X 8.568, Y -18.006, Z 101.150} C_DIS
   LIN {X 8.083, Y -19.784, Z 101.150} C_DIS
   LIN {X 7.965, Y -20.222, Z 101.150} C_DIS
   LIN {X 7.655, Y -20.586, Z 101.150} C_DIS
   LIN {X 6.567, Y -21.856, Z 101.150} C_DIS
   LIN {X 4.912, Y -22.615, Z 101.150} C_DIS
   LIN {X 4.590, Y -22.761, Z 101.150} C_DIS
   LIN {X 4.067, Y -22.762, Z 101.150} C_DIS
   LIN {X 2.479, Y -22.769, Z 101.150} C_DIS
   LIN {X 1.496, Y -22.329, Z 101.150} C_DIS
   LIN {X 0.594, Y -21.921, Z 101.150} C_DIS
   LIN {X -0.275, Y -20.948, Z 101.150} C_DIS
   LIN {X -0.796, Y -20.369, Z 101.150} C_DIS
   LIN {X -1.009, Y -19.692, Z 101.150} C_DIS
   LIN {X -1.419, Y -18.378, Z 101.150} C_DIS
   LIN {X -0.942, Y -16.267, Z 101.150} C_DIS
   LIN {X -0.738, Y -15.341, Z 101.150} C_DIS
   LIN {X -0.277, Y -14.824, Z 101.150} C_DIS
   LIN {X 0.603, Y -13.848, Z 101.150} C_DIS
   LIN {X 1.435, Y -13.472, Z 101.150} C_DIS
   LIN {X 2.518, Y -12.979, Z 101.150} C_DIS
   LIN {X 4.639, Y -12.965, Z 101.150} C_DIS
   LIN {X 4.931, Y -13.099, Z 101.150} C_DIS
   LIN {X 6.574, Y -13.845, Z 101.150} C_DIS
   LIN {X 8.097, Y -15.761, Z 101.150} C_DIS
   LIN {X 8.156, Y -15.835, Z 101.150}
   LaserEnd_Ext()
   LIN {X -2.825, Y -24.283, Z 101.150}
   LaserStart_Ext()
   LIN {X -2.985, Y -24.058, Z 101.150} C_DIS
   LIN {X -4.537, Y -21.896, Z 101.150} C_DIS
   LIN {X -5.336, Y -18.728, Z 101.150} C_DIS
   LIN {X -5.448, Y -18.300, Z 101.150} C_DIS
   LIN {X -5.369, Y -17.702, Z 101.150} C_DIS
   LIN {X -5.023, Y -15.158, Z 101.150} C_DIS
   LIN {X -4.394, Y -13.081, Z 101.150} C_DIS
   LIN {X -4.137, Y -12.200, Z 101.150} C_DIS
   LIN {X -3.024, Y -7.573, Z 101.150} C_DIS
   LIN {X -2.997, Y -7.453, Z 101.150} C_DIS
   LIN {X -1.870, Y 0.013, Z 101.150} C_DIS
   LIN {X -1.551, Y 8.639, Z 101.150} C_DIS
   LIN {X -1.540, Y 8.926, Z 101.150} C_DIS
   LIN {X -1.562, Y 9.176, Z 101.150} C_DIS
   LIN {X -2.439, Y 18.688, Z 101.150} C_DIS
   LIN {X -2.528, Y 19.141, Z 101.150} C_DIS
   LIN {X -2.843, Y 20.518, Z 101.150} C_DIS
   LIN {X -4.178, Y 26.634, Z 101.150} C_DIS
   LIN {X -4.644, Y 28.229, Z 101.150} C_DIS
   LIN {X -6.215, Y 32.793, Z 101.150} C_DIS
   LIN {X -6.958, Y 34.784, Z 101.150} C_DIS
   LIN {X -7.094, Y 35.104, Z 101.150} C_DIS
   LIN {X -7.300, Y 35.592, Z 101.150} C_DIS
   LIN {X -7.629, Y 36.371, Z 101.150} C_DIS
   LIN {X -8.225, Y 37.684, Z 101.150} C_DIS
   LIN {X -8.594, Y 38.492, Z 101.150} C_DIS
   LIN {X -8.978, Y 39.277, Z 101.150} C_DIS
   LIN {X -9.296, Y 39.929, Z 101.150} C_DIS
   LIN {X -9.462, Y 40.262, Z 101.150} C_DIS
   LIN {X -9.856, Y 41.047, Z 101.150} C_DIS
   LIN {X -10.274, Y 42.304, Z 101.150} C_DIS
   LIN {X -10.184, Y 43.951, Z 101.150} C_DIS
   LIN {X -9.425, Y 45.409, Z 101.150} C_DIS
   LIN {X -7.194, Y 46.787, Z 101.150} C_DIS
   LIN {X -6.150, Y 46.779, Z 101.150} C_DIS
   LIN {X -5.449, Y 46.774, Z 101.150} C_DIS
   LIN {X -5.059, Y 46.588, Z 101.150} C_DIS
   LIN {X -3.880, Y 46.023, Z 101.150} C_DIS
   LIN {X -2.938, Y 44.957, Z 101.150} C_DIS
   LIN {X -2.875, Y 44.866, Z 101.150} C_DIS
   LIN {X -2.154, Y 43.631, Z 101.150} C_DIS
   LIN {X -1.382, Y 42.265, Z 101.150} C_DIS
   LIN {X -1.043, Y 41.662, Z 101.150} C_DIS
   LIN {X -0.652, Y 40.925, Z 101.150} C_DIS
   LIN {X 0.561, Y 38.643, Z 101.150} C_DIS
   LIN {X 2.071, Y 35.395, Z 101.150} C_DIS
   LIN {X 3.610, Y 32.166, Z 101.150} C_DIS
   LIN {X 6.149, Y 25.775, Z 101.150} C_DIS
   LIN {X 6.196, Y 25.659, Z 101.150} C_DIS
   LIN {X 6.482, Y 24.787, Z 101.150} C_DIS
   LIN {X 8.224, Y 19.478, Z 101.150} C_DIS
   LIN {X 8.350, Y 18.979, Z 101.150} C_DIS
   LIN {X 10.507, Y 10.374, Z 101.150} C_DIS
   LIN {X 11.635, Y 3.479, Z 101.150} C_DIS
   LIN {X 11.921, Y 1.725, Z 101.150} C_DIS
   LIN {X 12.182, Y -0.919, Z 101.150} C_DIS
   LIN {X 12.435, Y -3.441, Z 101.150} C_DIS
   LIN {X 12.587, Y -6.231, Z 101.150} C_DIS
   LIN {X 12.698, Y -8.311, Z 101.150} C_DIS
   LIN {X 12.735, Y -10.945, Z 101.150} C_DIS
   LIN {X 12.754, Y -12.115, Z 101.150} C_DIS
   LIN {X 12.749, Y -12.558, Z 101.150} C_DIS
   LIN {X 12.707, Y -15.075, Z 101.150} C_DIS
   LIN {X 12.606, Y -17.441, Z 101.150} C_DIS
   LIN {X 12.562, Y -18.334, Z 101.150} C_DIS
   LIN {X 12.275, Y -19.585, Z 101.150} C_DIS
   LIN {X 11.907, Y -21.221, Z 101.150} C_DIS
   LIN {X 11.088, Y -22.425, Z 101.150} C_DIS
   LIN {X 9.713, Y -24.418, Z 101.150} C_DIS
   LIN {X 7.257, Y -26.057, Z 101.150} C_DIS
   LIN {X 7.119, Y -26.113, Z 101.150} C_DIS
   LIN {X 1.700, Y -26.590, Z 101.150} C_DIS
   LIN {X 0.476, Y -26.366, Z 101.150} C_DIS
   LIN {X -2.533, Y -24.472, Z 101.150} C_DIS
   LIN {X -2.825, Y -24.283, Z 101.150}
   LaserEnd_Ext()
   LIN {X -8.280, Y 44.955, Z 101.150}
   LaserStart_Ext()
   LIN {X -8.280, Y 40.127, Z 101.150}
   LaserEnd_Ext()
   LIN {X -7.280, Y 38.021, Z 101.150}
   LaserStart_Ext()
   LIN {X -7.280, Y 45.564, Z 101.150}
   LaserEnd_Ext()
   LIN {X -6.280, Y 45.780, Z 101.150}
   LaserStart_Ext()
   LIN {X -6.280, Y 35.747, Z 101.150}
   LaserEnd_Ext()
   LIN {X -5.280, Y 33.148, Z 101.150}
   LaserStart_Ext()
   LIN {X -5.280, Y 45.585, Z 101.150}
   LaserEnd_Ext()
   LIN {X -4.280, Y 44.965, Z 101.150}
   LaserStart_Ext()
   LIN {X -4.280, Y 30.244, Z 101.150}
   LaserEnd_Ext()
   LIN {X -4.280, Y -17.116, Z 101.150}
   LaserStart_Ext()
   LIN {X -4.280, Y -18.827, Z 101.150}
   LaserEnd_Ext()
   LIN {X -3.280, Y -21.932, Z 101.150}
   LaserStart_Ext()
   LIN {X -3.280, Y -12.832, Z 101.150}
   LaserEnd_Ext()
   LIN {X -3.280, Y 27.126, Z 101.150}
   LaserStart_Ext()
   LIN {X -3.280, Y 43.576, Z 101.150}
   LaserEnd_Ext()
   LIN {X -2.280, Y 41.821, Z 101.150}
   LaserStart_Ext()
   LIN {X -2.280, Y 22.627, Z 101.150}
   LaserEnd_Ext()
   LIN {X -2.280, Y -8.755, Z 101.150}
   LaserStart_Ext()
   LIN {X -2.280, Y -17.651, Z 101.150}
   LaserEnd_Ext()
   LIN {X -2.280, Y -18.976, Z 101.150}
   LaserStart_Ext()
   LIN {X -2.280, Y -23.326, Z 101.150}
   LaserEnd_Ext()
   LIN {X -1.280, Y -24.079, Z 101.150}
   LaserStart_Ext()
   LIN {X -1.280, Y -21.326, Z 101.150}
   LaserEnd_Ext()
   LIN {X -1.280, Y -14.446, Z 101.150}
   LaserStart_Ext()
   LIN {X -1.280, Y -2.780, Z 101.150}
   LaserEnd_Ext()
   LIN {X -1.280, Y 17.010, Z 101.150}
   LaserStart_Ext()
   LIN {X -1.280, Y 39.976, Z 101.150}
   LaserEnd_Ext()
   LIN {X -0.280, Y 38.079, Z 101.150}
   LaserStart_Ext()
   LIN {X -0.280, Y -13.334, Z 101.150}
   LaserEnd_Ext()
   LIN {X -0.280, Y -22.443, Z 101.150}
   LaserStart_Ext()
   LIN {X -0.280, Y -24.709, Z 101.150}
   LaserEnd_Ext()
   LIN {X 0.720, Y -25.338, Z 101.150}
   LaserStart_Ext()
   LIN {X 0.720, Y -23.075, Z 101.150}
   LaserEnd_Ext()
   LIN {X 0.720, Y -12.698, Z 101.150}
   LaserStart_Ext()
   LIN {X 0.720, Y 35.928, Z 101.150}
   LaserEnd_Ext()
   LIN {X 1.720, Y 33.807, Z 101.150}
   LaserStart_Ext()
   LIN {X 1.720, Y -12.244, Z 101.150}
   LaserEnd_Ext()
   LIN {X 1.720, Y -23.525, Z 101.150}
   LaserStart_Ext()
   LIN {X 1.720, Y -25.577, Z 101.150}
   LaserEnd_Ext()
   LIN {X 2.720, Y -25.497, Z 101.150}
   LaserStart_Ext()
   LIN {X 2.720, Y -23.768, Z 101.150}
   LaserEnd_Ext()
   LIN {X 2.720, Y -11.978, Z 101.150}
   LaserStart_Ext()
   LIN {X 2.720, Y 31.698, Z 101.150}
   LaserEnd_Ext()
   LIN {X 3.720, Y 29.180, Z 101.150}
   LaserStart_Ext()
   LIN {X 3.720, Y -11.971, Z 101.150}
   LaserEnd_Ext()
   LIN {X 3.720, Y -23.764, Z 101.150}
   LaserStart_Ext()
   LIN {X 3.720, Y -25.409, Z 101.150}
   LaserEnd_Ext()
   LIN {X 4.720, Y -25.321, Z 101.150}
   LaserStart_Ext()
   LIN {X 4.720, Y -23.752, Z 101.150}
   LaserEnd_Ext()
   LIN {X 4.720, Y -11.969, Z 101.150}
   LaserStart_Ext()
   LIN {X 4.720, Y 26.663, Z 101.150}
   LaserEnd_Ext()
   LIN {X 5.720, Y 23.900, Z 101.150}
   LaserStart_Ext()
   LIN {X 5.720, Y -12.359, Z 101.150}
   LaserEnd_Ext()
   LIN {X 5.720, Y -23.345, Z 101.150}
   LaserStart_Ext()
   LIN {X 5.720, Y -25.233, Z 101.150}
   LaserEnd_Ext()
   LIN {X 6.720, Y -25.145, Z 101.150}
   LaserStart_Ext()
   LIN {X 6.720, Y -22.886, Z 101.150}
   LaserEnd_Ext()
   LIN {X 6.720, Y -12.813, Z 101.150}
   LaserStart_Ext()
   LIN {X 6.720, Y 20.853, Z 101.150}
   LaserEnd_Ext()
   LIN {X 7.720, Y 17.379, Z 101.150}
   LaserStart_Ext()
   LIN {X 7.720, Y -13.680, Z 101.150}
   LaserEnd_Ext()
   LIN {X 7.720, Y -22.048, Z 101.150}
   LaserStart_Ext()
   LIN {X 7.720, Y -24.546, Z 101.150}
   LaserEnd_Ext()
   LIN {X 8.720, Y -23.878, Z 101.150}
   LaserStart_Ext()
   LIN {X 8.720, Y -20.877, Z 101.150}
   LaserEnd_Ext()
   LIN {X 8.720, Y -14.937, Z 101.150}
   LaserStart_Ext()
   LIN {X 8.720, Y 13.390, Z 101.150}
   LaserEnd_Ext()
   LIN {X 9.720, Y 8.989, Z 101.150}
   LaserStart_Ext()
   LIN {X 9.720, Y -22.646, Z 101.150}
   LaserEnd_Ext()
   LIN {X 10.720, Y -21.188, Z 101.150}
   LaserStart_Ext()
   LIN {X 10.720, Y 2.874, Z 101.150}
   LaserEnd_Ext()
   LIN {X 11.720, Y -9.920, Z 101.150}
   LaserStart_Ext()
   LIN {X 11.720, Y -14.266, Z 101.150}
   LaserEnd_Ext()
   LIN {X 8.232, Y -15.766, Z 102.000}
   LaserStart_Ext()
   LIN {X 8.480, Y -17.045, Z 102.000} C_DIS
   LIN {X 8.649, Y -17.936, Z 102.000} C_DIS
   LIN {X 8.457, Y -18.642, Z 102.000} C_DIS
   LIN {X 8.047, Y -20.160, Z 102.000} C_DIS
   LIN {X 6.975, Y -21.424, Z 102.000} C_DIS
   LIN {X 6.666, Y -21.784, Z 102.000} C_DIS
   LIN {X 5.961, Y -22.107, Z 102.000} C_DIS
   LIN {X 4.681, Y -22.700, Z 102.000} C_DIS
   LIN {X 3.785, Y -22.708, Z 102.000} C_DIS
   LIN {X 2.572, Y -22.713, Z 102.000} C_DIS
   LIN {X 1.015, Y -22.015, Z 102.000} C_DIS
   LIN {X 0.685, Y -21.869, Z 102.000} C_DIS
   LIN {X 0.503, Y -21.667, Z 102.000} C_DIS
   LIN {X -0.709, Y -20.320, Z 102.000} C_DIS
   LIN {X -1.301, Y -18.443, Z 102.000} C_DIS
   LIN {X -1.337, Y -18.331, Z 102.000} C_DIS
   LIN {X -1.303, Y -18.176, Z 102.000} C_DIS
   LIN {X -0.668, Y -15.300, Z 102.000} C_DIS
   LIN {X 0.675, Y -13.796, Z 102.000} C_DIS
   LIN {X 1.088, Y -13.610, Z 102.000} C_DIS
   LIN {X 2.610, Y -12.918, Z 102.000} C_DIS
   LIN {X 4.709, Y -12.903, Z 102.000} C_DIS
   LIN {X 5.898, Y -13.440, Z 102.000} C_DIS
   LIN {X 6.645, Y -13.779, Z 102.000} C_DIS
   LIN {X 7.175, Y -14.446, Z 102.000} C_DIS
   LIN {X 8.232, Y -15.766, Z 102.000}
   LaserEnd_Ext()
   LIN {X -2.394, Y 18.438, Z 102.000}
   LaserStart_Ext()
   LIN {X -2.606, Y 19.510, Z 102.000} C_DIS
   LIN {X -3.349, Y 22.761, Z 102.000} C_DIS
   LIN {X -4.220, Y 26.752, Z 102.000} C_DIS
   LIN {X -4.524, Y 27.793, Z 102.000} C_DIS
   LIN {X -6.418, Y 33.295, Z 102.000} C_DIS
   LIN {X -6.870, Y 34.507, Z 102.000} C_DIS
   LIN {X -6.953, Y 34.702, Z 102.000} C_DIS
   LIN {X -7.079, Y 34.999, Z 102.000} C_DIS
   LIN {X -7.510, Y 36.020, Z 102.000} C_DIS
   LIN {X -7.774, Y 36.624, Z 102.000} C_DIS
   LIN {X -8.642, Y 38.523, Z 102.000} C_DIS
   LIN {X -8.954, Y 39.161, Z 102.000} C_DIS
   LIN {X -9.347, Y 39.959, Z 102.000} C_DIS
   LIN {X -9.834, Y 40.924, Z 102.000} C_DIS
   LIN {X -9.910, Y 41.076, Z 102.000} C_DIS
   LIN {X -9.950, Y 41.195, Z 102.000} C_DIS
   LIN {X -10.339, Y 42.358, Z 102.000} C_DIS
   LIN {X -10.252, Y 43.828, Z 102.000} C_DIS
   LIN {X -10.243, Y 43.980, Z 102.000} C_DIS
   LIN {X -10.164, Y 44.131, Z 102.000} C_DIS
   LIN {X -9.444, Y 45.502, Z 102.000} C_DIS
   LIN {X -8.075, Y 46.334, Z 102.000} C_DIS
   LIN {X -7.261, Y 46.821, Z 102.000} C_DIS
   LIN {X -6.483, Y 46.819, Z 102.000} C_DIS
   LIN {X -5.516, Y 46.813, Z 102.000} C_DIS
   LIN {X -4.161, Y 46.167, Z 102.000} C_DIS
   LIN {X -3.946, Y 46.065, Z 102.000} C_DIS
   LIN {X -3.846, Y 45.954, Z 102.000} C_DIS
   LIN {X -2.970, Y 44.964, Z 102.000} C_DIS
   LIN {X -2.320, Y 43.860, Z 102.000} C_DIS
   LIN {X -2.218, Y 43.685, Z 102.000} C_DIS
   LIN {X -1.980, Y 43.265, Z 102.000} C_DIS
   LIN {X -1.027, Y 41.581, Z 102.000} C_DIS
   LIN {X -0.601, Y 40.782, Z 102.000} C_DIS
   LIN {X 0.639, Y 38.449, Z 102.000} C_DIS
   LIN {X 1.632, Y 36.313, Z 102.000} C_DIS
   LIN {X 3.530, Y 32.333, Z 102.000} C_DIS
   LIN {X 5.424, Y 27.564, Z 102.000} C_DIS
   LIN {X 6.052, Y 26.020, Z 102.000} C_DIS
   LIN {X 6.247, Y 25.535, Z 102.000} C_DIS
   LIN {X 8.190, Y 19.606, Z 102.000} C_DIS
   LIN {X 8.311, Y 19.239, Z 102.000} C_DIS
   LIN {X 8.639, Y 17.902, Z 102.000} C_DIS
   LIN {X 10.586, Y 10.135, Z 102.000} C_DIS
   LIN {X 11.889, Y 2.167, Z 102.000} C_DIS
   LIN {X 11.971, Y 1.666, Z 102.000} C_DIS
   LIN {X 12.046, Y 0.909, Z 102.000} C_DIS
   LIN {X 12.508, Y -3.686, Z 102.000} C_DIS
   LIN {X 12.746, Y -8.065, Z 102.000} C_DIS
   LIN {X 12.756, Y -8.231, Z 102.000} C_DIS
   LIN {X 12.762, Y -8.496, Z 102.000} C_DIS
   LIN {X 12.820, Y -12.035, Z 102.000} C_DIS
   LIN {X 12.802, Y -13.733, Z 102.000} C_DIS
   LIN {X 12.780, Y -14.995, Z 102.000} C_DIS
   LIN {X 12.670, Y -17.577, Z 102.000} C_DIS
   LIN {X 12.643, Y -18.254, Z 102.000} C_DIS
   LIN {X 12.571, Y -18.582, Z 102.000} C_DIS
   LIN {X 11.995, Y -21.143, Z 102.000} C_DIS
   LIN {X 10.324, Y -23.598, Z 102.000} C_DIS
   LIN {X 9.808, Y -24.345, Z 102.000} C_DIS
   LIN {X 8.828, Y -25.000, Z 102.000} C_DIS
   LIN {X 7.277, Y -26.038, Z 102.000} C_DIS
   LIN {X 3.669, Y -26.204, Z 102.000} C_DIS
   LIN {X 1.149, Y -26.425, Z 102.000} C_DIS
   LIN {X 0.610, Y -26.327, Z 102.000} C_DIS
   LIN {X -1.064, Y -25.273, Z 102.000} C_DIS
   LIN {X -2.731, Y -24.239, Z 102.000} C_DIS
   LIN {X -3.252, Y -23.522, Z 102.000} C_DIS
   LIN {X -4.448, Y -21.856, Z 102.000} C_DIS
   LIN {X -4.959, Y -19.828, Z 102.000} C_DIS
   LIN {X -5.367, Y -18.262, Z 102.000} C_DIS
   LIN {X -5.078, Y -16.068, Z 102.000} C_DIS
   LIN {X -4.949, Y -15.118, Z 102.000} C_DIS
   LIN {X -4.714, Y -14.343, Z 102.000} C_DIS
   LIN {X -4.013, Y -11.940, Z 102.000} C_DIS
   LIN {X -3.195, Y -8.537, Z 102.000} C_DIS
   LIN {X -2.963, Y -7.520, Z 102.000} C_DIS
   LIN {X -2.841, Y -6.760, Z 102.000} C_DIS
   LIN {X -1.868, Y -0.309, Z 102.000} C_DIS
   LIN {X -1.578, Y 7.516, Z 102.000} C_DIS
   LIN {X -1.513, Y 8.687, Z 102.000} C_DIS
   LIN {X -1.563, Y 9.418, Z 102.000} C_DIS
   LIN {X -2.394, Y 18.438, Z 102.000}
   LaserEnd_Ext()
   LIN {X 0.952, Y -25.360, Z 102.000}
   LaserStart_Ext()
   LIN {X 1.848, Y -25.360, Z 102.000}
   LaserEnd_Ext()
   LIN {X 7.985, Y -24.360, Z 102.000}
   LaserStart_Ext()
   LIN {X -0.638, Y -24.360, Z 102.000}
   LaserEnd_Ext()
   LIN {X -2.133, Y -23.360, Z 102.000}
   LaserStart_Ext()
   LIN {X 1.571, Y -23.360, Z 102.000}
   LaserEnd_Ext()
   LIN {X 5.635, Y -23.360, Z 102.000}
   LaserStart_Ext()
   LIN {X 9.273, Y -23.360, Z 102.000}
   LaserEnd_Ext()
   LIN {X 9.957, Y -22.360, Z 102.000}
   LaserStart_Ext()
   LIN {X 7.489, Y -22.360, Z 102.000}
   LaserEnd_Ext()
   LIN {X -0.219, Y -22.360, Z 102.000}
   LaserStart_Ext()
   LIN {X -2.855, Y -22.360, Z 102.000}
   LaserEnd_Ext()
   LIN {X -3.541, Y -21.360, Z 102.000}
   LaserStart_Ext()
   LIN {X -1.119, Y -21.360, Z 102.000}
   LaserEnd_Ext()
   LIN {X 8.340, Y -21.360, Z 102.000}
   LaserStart_Ext()
